fbBahn_Roll1.IsPosi_Aktiv_VonBahn:= fbGeberHandling_VonBahn_Roll1.OsAktiv;
fbBahn_Roll1.IsPosi_Fertig_VonBahn:= fbGeberHandling_VonBahn_Roll1.OsFertig
							OR	bI_AbbruchPosi_VonBahn_Roll1
								AND ( fbBahn_Roll1.SKet2 = 314
									OR	fbBahn_Roll1.SKet2 = 354
									OR	fbBahn_Roll1.SKet2 = 754
									OR	fbBahn_Roll1.SKet2 = 759 );

fbBahn_Roll1.IsLaderHatPlatteGeholt		:= strIO_GHdshk_Roll1.b_HatPlatteGeholt;
fbBahn_Roll1.IsLaderHatPlatteAbgelegt	:= strIO_GHdshk_Roll1.b_HatPlatteAbgelegt;
END_ACTION

ACTION D_Bahnjob_Riem1:
(*----------------------------------------------------------------------------------------------------------------------------------*)
(*----------------------------------------------------------------------------------------------------------------------------------*)
(*	Wenn das Bahnmodul den Job übernommen hat und der Job ausgeführt wird, muss der Job gelöscht werden					*)
(*----------------------------------------------------------------------------------------------------------------------------------*)
(*----------------------------------------------------------------------------------------------------------------------------------*)

fbBahn_Riem1.IwDoJob_AufBahn:= strIO_GHdshk_Riem1.str_DoJob_AufBahn;				(* Job Auf Bahn von der Struktur in den Baustein schreiben *)
fbBahn_Riem1.IwDoJob_VonBahn:= strIO_GHdshk_Riem1.str_DoJob_VonBahn;				(* Job Von Bahn von der Struktur in den Baustein schreiben *)
fbBahn_Riem1.IwAnzahlPlatten_BeiVonBahn := strIO_GHdshk_Riem1.i_AnzahlPlattenVonBahn;	(* Azahl der Platten in den Baustein geben *)

IF	fbBahn_Riem1.IwDoJob_AufBahn > eRolljobKeinJob							(* Wenn der Baustein den Job Auf Bahn ausführt, Job in der Struktur zurücksetzen *)
	AND	strIO_GHdshk_Riem1.str_JobAktiv_AufBahn = fbBahn_Riem1.IwDoJob_AufBahn		(* Aktiver Job in der Struktur angekommen *)
THEN
	strIO_GHdshk_Riem1.str_DoJob_AufBahn:= eRolljobKeinJob;
END_IF;

IF	fbBahn_Riem1.IwDoJob_VonBahn > eRolljobKeinJob							(* Wenn der Baustein den Job Auf Bahn ausführt, Job in der Struktur zurücksetzen *)
	AND	strIO_GHdshk_Riem1.str_JobAktiv_VonBahn = fbBahn_Riem1.IwDoJob_VonBahn		(* Aktiver Job in der Struktur angekommen *)
THEN
	strIO_GHdshk_Riem1.str_DoJob_VonBahn:= eRolljobKeinJob;
END_IF;


IF	(( fbBahn_Riem1.IsHand											(* Wenn Reset auf die Quellbahn gemacht wird, darf der Jobbaustein nicht buchen *)
		AND	fbBahn_Riem1.IsReset )
	OR	strIO_TrE.iReset <> 0 )
	AND NOT strIO_GHdshk_Riem1.b_JobVonBahnAbgebrochen
	AND 	strIO_GHdshk_Riem1.str_JobAktiv_VonBahn <> eRolljobKeinJob
	AND 	strIO_GHdshk_Riem1.str_JobAktiv_VonBahn <> eRolljobAnsBahnendeVorlauf
	AND 	strIO_GHdshk_Riem1.str_JobAktiv_VonBahn <> eRolljobAnBahnanfangRuecklauf
THEN
	strIO_GHdshk_Riem1.b_JobVonBahnAbgebrochen:= TRUE;
END_IF;
END_ACTION

ACTION D_Bahnjob_Riem2:
(*----------------------------------------------------------------------------------------------------------------------------------*)
(*----------------------------------------------------------------------------------------------------------------------------------*)
(*	Wenn das Bahnmodul den Job übernommen hat und der Job ausgeführt wird, muss der Job gelöscht werden					*)
(*----------------------------------------------------------------------------------------------------------------------------------*)
(*----------------------------------------------------------------------------------------------------------------------------------*)

fbBahn_Riem2.IwDoJob_AufBahn:= strIO_GHdshk_Riem2.str_DoJob_AufBahn;				(* Job Auf Bahn von der Struktur in den Baustein schreiben *)
fbBahn_Riem2.IwDoJob_VonBahn:= strIO_GHdshk_Riem2.str_DoJob_VonBahn;				(* Job Von Bahn von der Struktur in den Baustein schreiben *)
fbBahn_Riem2.IwAnzahlPlatten_BeiVonBahn := strIO_GHdshk_Riem2.i_AnzahlPlattenVonBahn;	(* Azahl der Platten in den Baustein geben *)

IF	fbBahn_Riem2.IwDoJob_AufBahn > eRolljobKeinJob							(* Wenn der Baustein den Job Auf Bahn ausführt, Job in der Struktur zurücksetzen *)
	AND	strIO_GHdshk_Riem2.str_JobAktiv_AufBahn = fbBahn_Riem2.IwDoJob_AufBahn		(* Aktiver Job in der Struktur angekommen *)
THEN
	strIO_GHdshk_Riem2.str_DoJob_AufBahn:= eRolljobKeinJob;
END_IF;

IF	fbBahn_Riem2.IwDoJob_VonBahn > eRolljobKeinJob							(* Wenn der Baustein den Job Auf Bahn ausführt, Job in der Struktur zurücksetzen *)
	AND	strIO_GHdshk_Riem2.str_JobAktiv_VonBahn = fbBahn_Riem2.IwDoJob_VonBahn		(* Aktiver Job in der Struktur angekommen *)
THEN
	strIO_GHdshk_Riem2.str_DoJob_VonBahn:= eRolljobKeinJob;
END_IF;


IF	(( fbBahn_Riem2.IsHand											(* Wenn Reset auf die Quellbahn gemacht wird, darf der Jobbaustein nicht buchen *)
		AND	fbBahn_Riem2.IsReset )
	OR	strIO_TrE.iReset <> 0 )
	AND NOT strIO_GHdshk_Riem2.b_JobVonBahnAbgebrochen
	AND 	strIO_GHdshk_Riem2.str_JobAktiv_VonBahn <> eRolljobKeinJob
	AND 	strIO_GHdshk_Riem2.str_JobAktiv_VonBahn <> eRolljobAnsBahnendeVorlauf
	AND 	strIO_GHdshk_Riem2.str_JobAktiv_VonBahn <> eRolljobAnBahnanfangRuecklauf
THEN
	strIO_GHdshk_Riem2.b_JobVonBahnAbgebrochen:= TRUE;
END_IF;
END_ACTION

ACTION D_Bahnjob_Roll1:
(*----------------------------------------------------------------------------------------------------------------------------------*)
(*----------------------------------------------------------------------------------------------------------------------------------*)
(*	Wenn das Bahnmodul den Job übernommen hat und der Job ausgeführt wird, muss der Job gelöscht werden					*)
(*----------------------------------------------------------------------------------------------------------------------------------*)
(*----------------------------------------------------------------------------------------------------------------------------------*)

fbBahn_Roll1.IwDoJob_AufBahn:= strIO_GHdshk_Roll1.str_DoJob_AufBahn;				(* Job Auf Bahn von der Struktur in den Baustein schreiben *)
fbBahn_Roll1.IwDoJob_VonBahn:= strIO_GHdshk_Roll1.str_DoJob_VonBahn;				(* Job Von Bahn von der Struktur in den Baustein schreiben *)
fbBahn_Roll1.IwAnzahlPlatten_BeiVonBahn:= strIO_GHdshk_Roll1.i_AnzahlPlattenVonBahn;	(* Azahl der Platten in den Baustein geben *)

IF	fbBahn_Roll1.IwDoJob_AufBahn > eRolljobKeinJob							(* Wenn der Baustein den Job Auf Bahn ausführt, Job in der Struktur zurücksetzen *)
	AND	strIO_GHdshk_Roll1.str_JobAktiv_AufBahn = fbBahn_Roll1.IwDoJob_AufBahn		(* Aktiver Job in der Struktur angekommen *)
THEN
	strIO_GHdshk_Roll1.str_DoJob_AufBahn:= eRolljobKeinJob;
END_IF;

IF	fbBahn_Roll1.IwDoJob_VonBahn > eRolljobKeinJob							(* Wenn der Baustein den Job Auf Bahn ausführt, Job in der Struktur zurücksetzen *)
	AND	strIO_GHdshk_Roll1.str_JobAktiv_VonBahn = fbBahn_Roll1.IwDoJob_VonBahn		(* Aktiver Job in der Struktur angekommen *)
THEN
	strIO_GHdshk_Roll1.str_DoJob_VonBahn:= eRolljobKeinJob;
END_IF;


IF	(( fbBahn_Roll1.IsHand											(* Wenn Reset auf die Quellbahn gemacht wird, darf der Jobbaustein nicht buchen *)
		AND	fbBahn_Roll1.IsReset )
	OR	strIO_TrE.iReset <> 0 )
	AND NOT strIO_GHdshk_Roll1.b_JobVonBahnAbgebrochen
	AND 	strIO_GHdshk_Roll1.str_JobAktiv_VonBahn <> eRolljobKeinJob
	AND 	strIO_GHdshk_Roll1.str_JobAktiv_VonBahn <> eRolljobAnsBahnendeVorlauf
	AND 	strIO_GHdshk_Roll1.str_JobAktiv_VonBahn <> eRolljobAnBahnanfangRuecklauf
THEN
	strIO_GHdshk_Roll1.b_JobVonBahnAbgebrochen:= TRUE;
END_IF;
END_ACTION

ACTION E_Ausgaenge_Hub:
(*----------------------------------------------------------------------------------------------------------------------------------*)
(*----------------------------------------------------------------------------------------------------------------------------------*)
(*                 Ausgänge Hub Winkeluebergabe															*)
(*----------------------------------------------------------------------------------------------------------------------------------*)
(*----------------------------------------------------------------------------------------------------------------------------------*)

IF	bI_Automatik
THEN
	IF	strIO_GHdshk_Riem1.b_SektionenKoppelnInY
	THEN
		bQ_Sektion1AS:= bQ_Sektion2AS;
		bQ_Sektion1GS:= bQ_Sektion2GS;

	ELSIF	fbBahn_Roll1.OwBahnStatus = iAutomatikAktivJob
	THEN
		IF	bI_HebenSenkenInvers
		THEN
			bQ_Sektion1AS:= fbBahn_Roll1.OsBahnAufFoerderhoehe;
			bQ_Sektion1GS:= NOT fbBahn_Roll1.OsBahnAufFoerderhoehe;
		ELSE
			bQ_Sektion1AS:= NOT fbBahn_Roll1.OsBahnAufFoerderhoehe;
			bQ_Sektion1GS:= fbBahn_Roll1.OsBahnAufFoerderhoehe;
		END_IF;

	ELSIF	fbBahn_Riem1.OwBahnStatus = iAutomatikAktivJob
	THEN
		IF	bI_HebenSenkenInvers
		THEN
			bQ_Sektion1AS:= NOT fbBahn_Riem1.OsBahnAufFoerderhoehe;
			bQ_Sektion1GS:= fbBahn_Riem1.OsBahnAufFoerderhoehe;
		ELSE
			bQ_Sektion1AS:= fbBahn_Riem1.OsBahnAufFoerderhoehe;
			bQ_Sektion1GS:= NOT fbBahn_Riem1.OsBahnAufFoerderhoehe;
		END_IF;
	END_IF;

	IF	strIO_GHdshk_Riem2.b_SektionenKoppelnInY
	THEN
		bQ_Sektion2AS:= bQ_Sektion1AS;
		bQ_Sektion2GS:= bQ_Sektion1GS;

	ELSIF	fbBahn_Roll1.OwBahnStatus = iAutomatikAktivJob
	THEN
		IF	bI_HebenSenkenInvers
		THEN
			bQ_Sektion2AS:= fbBahn_Roll1.OsBahnAufFoerderhoehe;
			bQ_Sektion2GS:= NOT fbBahn_Roll1.OsBahnAufFoerderhoehe;
		ELSE
			bQ_Sektion2AS:= NOT fbBahn_Roll1.OsBahnAufFoerderhoehe;
			bQ_Sektion2GS:= fbBahn_Roll1.OsBahnAufFoerderhoehe;
		END_IF;

	ELSIF	fbBahn_Riem2.OwBahnStatus = iAutomatikAktivJob
	THEN
		IF	bI_HebenSenkenInvers
		THEN
			bQ_Sektion2AS:= NOT fbBahn_Riem2.OsBahnAufFoerderhoehe;
			bQ_Sektion2GS:= fbBahn_Riem2.OsBahnAufFoerderhoehe;
		ELSE
			bQ_Sektion2AS:= fbBahn_Riem2.OsBahnAufFoerderhoehe;
			bQ_Sektion2GS:= NOT fbBahn_Riem2.OsBahnAufFoerderhoehe;
		END_IF;
	END_IF;

	IF	fbBahn_Roll1.OwBahnStatus = iAutomatikBereitJob
		AND	fbBahn_Riem1.OwBahnStatus = iAutomatikBereitJob
		AND	fbBahn_Riem2.OwBahnStatus = iAutomatikBereitJob
		AND NOT strIO_GHdshk_Roll1.b_BahnBelegt
		AND NOT strIO_GHdshk_Riem1.b_BahnBelegt
		AND NOT strIO_GHdshk_Riem2.b_BahnBelegt
		AND strIO_TrE.iAnzahlPlatten = 0
		AND strIO_TrE.asBarcode[1] = ''
	THEN
		IF	bI_HubGrundWennFrei_Sek_1
		THEN
			bQ_Sektion1AS:= FALSE;
			bQ_Sektion1GS:= TRUE;

		ELSIF bI_HubArbeitWennFrei_Sek_1
		THEN
			bQ_Sektion1AS:= TRUE;
			bQ_Sektion1GS:= FALSE;
		END_IF;

		IF	bI_HubGrundWennFrei_Sek_2
		THEN
			bQ_Sektion2AS:= FALSE;
			bQ_Sektion2GS:= TRUE;

		ELSIF bI_HubArbeitWennFrei_Sek_2
		THEN
			bQ_Sektion2AS:= TRUE;
			bQ_Sektion2GS:= FALSE;
		END_IF;

	ELSIF	fbBahn_Roll1.OwBahnStatus = iAutomatikBereitJob
		AND	fbBahn_Riem1.OwBahnStatus = iAutomatikBereitJob
		AND	fbBahn_Riem2.OwBahnStatus = iAutomatikBereitJob
		AND 	strIO_GHdshk_Roll1.b_BahnBelegt
		AND 	strIO_GHdshk_Riem1.b_BahnBelegt
		AND 	strIO_GHdshk_Riem2.b_BahnBelegt
		AND 	strIO_TrE.iAnzahlPlatten = 0
		AND 	strIO_TrE.asBarcode[1] = ''
	THEN
		IF	bI_HubGrundWennBelegt_Sek_1
		THEN
			bQ_Sektion1AS:= FALSE;
			bQ_Sektion1GS:= TRUE;

		ELSIF bI_HubArbeitWennBelegt_Sek_1
		THEN
			bQ_Sektion1AS:= TRUE;
			bQ_Sektion1GS:= FALSE;
		END_IF;

		IF	bI_HubGrundWennBelegt_Sek_2
		THEN
			bQ_Sektion2AS:= FALSE;
			bQ_Sektion2GS:= TRUE;

		ELSIF bI_HubArbeitWennBelegt_Sek_2
		THEN
			bQ_Sektion2AS:= TRUE;
			bQ_Sektion2GS:= FALSE;
		END_IF;
	END_IF;

	bHandHebenSenkenAktiv_Sek_1:= FALSE;
	bHandHebenSenkenAktiv_Sek_2:= FALSE;

ELSIF	bI_Hand
THEN
	IF	( strIO_GLmHand.bI_Heben
		OR	strIO_GLmHand.bI_Senken )
		AND	bI_FreigabeHandHebenSenkenSek1
	THEN
		bHandHebenSenkenAktiv_Sek_1:= TRUE;
	END_IF;

	IF	( strIO_GLmHand.bI_Heben
		OR	strIO_GLmHand.bI_Senken )
		AND	bI_FreigabeHandHebenSenkenSek2
	THEN
		bHandHebenSenkenAktiv_Sek_2:= TRUE;
	END_IF;

	IF	bHandHebenSenkenAktiv_Sek_1
	THEN
		bQ_Sektion1AS:= fbBahn_Roll1.OsBahnAufFoerderhoehe;
		bQ_Sektion1GS:= NOT fbBahn_Roll1.OsBahnAufFoerderhoehe;
	END_IF;

	IF	bHandHebenSenkenAktiv_Sek_2
	THEN
		bQ_Sektion2AS:= fbBahn_Roll1.OsBahnAufFoerderhoehe;
		bQ_Sektion2GS:= NOT fbBahn_Roll1.OsBahnAufFoerderhoehe;
	END_IF;

ELSE
	bHandHebenSenkenAktiv_Sek_1:= FALSE;
	bHandHebenSenkenAktiv_Sek_2:= FALSE;
END_IF;
END_ACTION

ACTION E_Ausgaenge_Riem1:
(*----------------------------------------------------------------------------------------------------------------------------------*)
(*----------------------------------------------------------------------------------------------------------------------------------*)
(*                 Ausgänge																											*)
(*----------------------------------------------------------------------------------------------------------------------------------*)
(*----------------------------------------------------------------------------------------------------------------------------------*)
fbRampe_Riem1(
	lrI_Acceleration:= strIO_GHdshk_Riem1.str_BahnRampen.lrBeschleunigung_mms2,
	lrI_Deceleration:= strIO_GHdshk_Riem1.str_BahnRampen.lrVerzoegerung_mms2,
	lrI_FastDeceleration:= strIO_GHdshk_Riem1.str_BahnRampen.lrNotverzoegerung_mms2,
	lrI_TimeBase:= lrZyklusZeit_SPS,
	lrI_MaxVelo:= strIO_GHdshk_Riem1.str_BahnSpeed.rVmaxSpeed,
	lrI_Velocity:= fbBahn_Riem1.OwBahnSpeed,
	lrI_CoupleVelocity:= fbBahn_Riem2.OwBahnSpeed,
	lrI_CoupleAcceleration:= strIO_GHdshk_Riem2.str_BahnRampen.lrBeschleunigung_mms2,
	lrI_CoupleDeceleration:= strIO_GHdshk_Riem2.str_BahnRampen.lrVerzoegerung_mms2,
	bI_Couple:= strIO_GHdshk_Riem1.b_SektionenKoppelnInY
			AND	bI_Automatik,
	bI_Enable:= bI_SicherheitOK,
	bI_ErrorQuit:= strIO_GLmHand.bI_QuittStoerung,
	lrQ_ActVelocity=> ,
	uiQ_ErrorNumber=> , 
	iQ_AnalogueValue=> ,
	bQ_TargetVelo=> , 
	bQ_Acceleration=> ,
	bQ_Deceleration=> ,
	bQ_MovePos=> , 
	bQ_MoveNeg=> , 
	bQ_MoveNot=> ,
	bQ_Error=> );

IF	fbRampe_Riem1.bQ_MovePos
THEN
	iBahnLetzteBewegung_Sek_1:= 11;

ELSIF	fbRampe_Riem1.bQ_MoveNeg
THEN
	iBahnLetzteBewegung_Sek_1:= 12;
END_IF;
END_ACTION

ACTION E_Ausgaenge_Riem2:
(*----------------------------------------------------------------------------------------------------------------------------------*)
(*----------------------------------------------------------------------------------------------------------------------------------*)
(*                 Ausgänge																											*)
(*----------------------------------------------------------------------------------------------------------------------------------*)
(*----------------------------------------------------------------------------------------------------------------------------------*)
fbRampe_Riem2(
	lrI_Acceleration:= strIO_GHdshk_Riem2.str_BahnRampen.lrBeschleunigung_mms2,
	lrI_Deceleration:= strIO_GHdshk_Riem2.str_BahnRampen.lrVerzoegerung_mms2,
	lrI_FastDeceleration:= strIO_GHdshk_Riem2.str_BahnRampen.lrNotverzoegerung_mms2,
	lrI_TimeBase:= lrZyklusZeit_SPS,
	lrI_MaxVelo:= strIO_GHdshk_Riem2.str_BahnSpeed.rVmaxSpeed,
	lrI_Velocity:= fbBahn_Riem2.OwBahnSpeed,
	lrI_CoupleVelocity:= fbBahn_Riem1.OwBahnSpeed,
	lrI_CoupleAcceleration:= strIO_GHdshk_Riem1.str_BahnRampen.lrBeschleunigung_mms2,
	lrI_CoupleDeceleration:= strIO_GHdshk_Riem1.str_BahnRampen.lrVerzoegerung_mms2,
	bI_Couple:= strIO_GHdshk_Riem2.b_SektionenKoppelnInY
			AND	bI_Automatik,
	bI_Enable:= bI_SicherheitOK,
	bI_ErrorQuit:= strIO_GLmHand.bI_QuittStoerung,
	lrQ_ActVelocity=> ,
	uiQ_ErrorNumber=> , 
	iQ_AnalogueValue=> ,
	bQ_TargetVelo=> , 
	bQ_Acceleration=> ,
	bQ_Deceleration=> ,
	bQ_MovePos=> ,
	bQ_MoveNeg=> ,
	bQ_MoveNot=> ,
	bQ_Error=> );

IF	fbRampe_Riem2.bQ_MovePos
THEN
	iBahnLetzteBewegung_Sek_2:= 11;

ELSIF	fbRampe_Riem2.bQ_MoveNeg
THEN
	iBahnLetzteBewegung_Sek_2:= 12;
END_IF;
END_ACTION

ACTION E_Ausgaenge_Roll1:
(*----------------------------------------------------------------------------------------------------------------------------------*)
(*----------------------------------------------------------------------------------------------------------------------------------*)
(*                 Ausgänge																											*)
(*----------------------------------------------------------------------------------------------------------------------------------*)
(*----------------------------------------------------------------------------------------------------------------------------------*)
fbRampe_Roll1(
	lrI_Acceleration:= strIO_GHdshk_Roll1.str_BahnRampen.lrBeschleunigung_mms2,
	lrI_Deceleration:= strIO_GHdshk_Roll1.str_BahnRampen.lrVerzoegerung_mms2,
	lrI_FastDeceleration:= strIO_GHdshk_Roll1.str_BahnRampen.lrNotverzoegerung_mms2,
	lrI_TimeBase:= lrZyklusZeit_SPS,
	lrI_MaxVelo:= strIO_GHdshk_Roll1.str_BahnSpeed.rVmaxSpeed,
	lrI_Velocity:= fbBahn_Roll1.OwBahnSpeed,
	lrI_CoupleVelocity:= 0,
	lrI_CoupleAcceleration:= 0,
	lrI_CoupleDeceleration:= 0,
	bI_Couple:= FALSE,
	bI_Enable:= bI_SicherheitOK,
	bI_ErrorQuit:= strIO_GLmHand.bI_QuittStoerung,
	lrQ_ActVelocity=> ,
	uiQ_ErrorNumber=> ,
	iQ_AnalogueValue=> ,
	bQ_TargetVelo=> , 
	bQ_Acceleration=> , 
	bQ_Deceleration=> ,
	bQ_MovePos=> ,
	bQ_MoveNeg=> , 
	bQ_MoveNot=> ,
	bQ_Error=> );

IF	fbRampe_Roll1.bQ_MovePos
THEN
	iBahnLetzteBewegung_Sek_1:= 1;
	iBahnLetzteBewegung_Sek_2:= 1;

ELSIF	fbRampe_Roll1.bQ_MoveNeg
THEN
	iBahnLetzteBewegung_Sek_1:= 2;
	iBahnLetzteBewegung_Sek_2:= 2;
END_IF;
END_ACTION

ACTION F_Positionierung_Riem1:
(*----------------------------------------------------------------------------------------------------------------------------------*)
(*----------------------------------------------------------------------------------------------------------------------------------*)
(*                 Positionierung																	*)
(*----------------------------------------------------------------------------------------------------------------------------------*)
(*----------------------------------------------------------------------------------------------------------------------------------*)


(*------ Achse Istwertsetzen  ---------------------------------*)
IF	uiI_AxId_Riem1 <> 0
THEN
	IF	fbBahn_Riem1.IwDoJob_AufBahn = eRolljobKeinJob
		AND	fbBahn_Riem1.OwJobAktiv_AufBahn = eRolljobKeinJob
		AND	fbBahn_Riem1.IwDoJob_VonBahn = eRolljobKeinJob
		AND	fbBahn_Riem1.OwJobAktiv_VonBahn = eRolljobKeinJob
		AND	fbAxIstwert_Riem1.OwOut.eAchsStatus = eStatAchse_BereitFuerJob
		AND NOT strIO_GHdshk_Riem1.b_BahnBelegt
		AND	strIO_TrE.iAnzahlPlatten = 0
		AND	strIO_TrE.asBarcode[1] = ''
		AND NOT bIstwertSetzen_Riem1
		AND ( AxFrNc_fPosIst[uiI_AxId_Riem1] > 50000
			OR	AxFrNc_fPosIst[uiI_AxId_Riem1] < -50000 )
	THEN
		bIstwertSetzen_Riem1:= TRUE;
	END_IF;

	fbAxIstwert_Riem1.AxId:= uiI_AxId_Riem1;
	fbAxIstwert_Riem1.IwResetMode:= 0;		(* Reset Modul *)

	fbAxIstwert_Riem1.IsHand:= bI_Hand;

	fbAxIstwert_Riem1.IsResetNachNotHalt:=
		AxFrNcFehler[uiI_AxId_Riem1]
		AND 	strIO_GLmHand.bI_QuittStoerung;

	fbAxIstwert_Riem1.IsAxFrNc_Auftraglaeuft:= AxFrNcAuftraglaeuft[uiI_AxId_Riem1];
	fbAxIstwert_Riem1.IsAxFrNc_Steht:= AxFrNcSteht[uiI_AxId_Riem1];
	fbAxIstwert_Riem1.IsAxFrNc_Geeicht:= AxFrNcGeeicht[uiI_AxId_Riem1];
	fbAxIstwert_Riem1.IsAxFrNc_Fehler:= AxFrNcFehler[uiI_AxId_Riem1];
	fbAxIstwert_Riem1.IwAxFrNc_nErrorCode:= AxFrNc_nErrorCode[uiI_AxId_Riem1];
	fbAxIstwert_Riem1.IsModuloAchse:= FALSE;
	
	fbAxIstwert_Riem1.IsReset:=
		( bI_FreigabeHandVorZurueck_Riem1
			OR	bI_FreigabeReset )
		AND	strIO_GLmHand.bI_Reset;
	
	IF	bIstwertSetzen_Riem1
		AND NOT fbAxIstwert_Riem1.IsIstwertSetzen
	THEN
		fbAxIstwert_Riem1.IsIstwertSetzen:= TRUE;
		fbAxIstwert_Riem1.IwWertIstwertSetzen:= 0;
	END_IF;
	
	IF	fbAxIstwert_Riem1.IsIstwertSetzen
		AND	fbAxIstwert_Riem1.OwOut.xIstwertGesetzt
	THEN
		fbAxIstwert_Riem1.IsIstwertSetzen:= FALSE;
		bIstwertSetzen_Riem1:= FALSE;
		lrIstwert_Bahn_Riem1:= 0;
	END_IF;


		fbAxIstwert_Riem1();

(*------ Simulation Istwert  ---------------------------------*)

	IF	bI_Testbetrieb
	THEN
		IF	strIO_GHdshk_Riem1.b_BahnVor
		THEN
			lrIstwert_Bahn_Riem1:=
				lrIstwert_Bahn_Riem1
				+ ABS((( strIO_GHdshk_Riem1.lr_Bahnspeed_Vorgabe * 1000) / 60 ) * lrZyklusZeit_SPS );
	
		ELSIF strIO_GHdshk_Riem1.b_BahnZurueck
		THEN
			lrIstwert_Bahn_Riem1:=
				lrIstwert_Bahn_Riem1
				- ABS((( strIO_GHdshk_Riem1.lr_Bahnspeed_Vorgabe * 1000) / 60 ) * lrZyklusZeit_SPS );
		END_IF;
	
		AxFrNc_fPosIst[uiI_AxId_Riem1]:= LREAL_TO_REAL ( lrIstwert_Bahn_Riem1 );
	END_IF;
END_IF;

IF ( bI_Testbetrieb
	OR	bI_OhneImpulsgeber_Riem1 )
	AND	uiI_AxId_Riem1 = 0
THEN
	fbVirtuellerImpulsgeber_Riem1(
		bI_Start:= strIO_GHdshk_Riem1.b_BahnVor
				OR	strIO_GHdshk_Riem1.b_BahnZurueck,
		lrI_TimeBase:= lrZyklusZeit_SPS,
		lrI_Speed:= ABS(strIO_GHdshk_Riem1.lr_Bahnspeed_Vorgabe),
		lrI_WegProImpuls:= strIO_GHdshk_Riem1.str_Bahndaten.rWegProImpuls,
		IO_Impulse:= iIncGeberZaehler_Riem1 );
END_IF;

(*------ AufBahn Positionierung Bahn  ---------------------------------*)
IF	uiI_AxId_Riem1 <> 0
THEN
	fbGeberHandling_AufBahn_Riem1.IwMode:= 1;		(* Achse auswerten *)
	fbGeberHandling_AufBahn_Riem1.IwIstwert:= AxFrNc_fPosIst[uiI_AxId_Riem1];
	fbGeberHandling_AufBahn_Riem1.IwIncGeberZaehler:= 0;
	fbGeberHandling_AufBahn_Riem1.IwWegProImpuls:= 0;
ELSE
	fbGeberHandling_AufBahn_Riem1.IwMode:= 2;		(* Zähler auswerten *)
	fbGeberHandling_AufBahn_Riem1.IwIstwert:= 0;
	fbGeberHandling_AufBahn_Riem1.IwIncGeberZaehler:= iIncGeberZaehler_Riem1;
	fbGeberHandling_AufBahn_Riem1.IwWegProImpuls:= strIO_GHdshk_Riem1.str_Bahndaten.rWegProImpuls;
END_IF;

fbGeberHandling_AufBahn_Riem1.IsAnfangBahn:= fbBahn_Riem1.IsAnfangBahn;
fbGeberHandling_AufBahn_Riem1.IsEndeBahn:= fbBahn_Riem1.IsEndeBahn;
fbGeberHandling_AufBahn_Riem1.IsStart:= fbBahn_Riem1.OsPosi_Start_AufBahn;
fbGeberHandling_AufBahn_Riem1.IsIncGeber:=  FALSE;
fbGeberHandling_AufBahn_Riem1.IsRestwertSchreiben:= TRUE;

fbGeberHandling_AufBahn_Riem1.IsIstwertGesetzt:= FALSE;
fbGeberHandling_AufBahn_Riem1.IsImRuecklauf:=
	fbBahn_Riem1.IwDoJob_AufBahn = eRolljobAufBahnPosiRuecklauf
	OR	fbBahn_Riem1.OwJobAktiv_AufBahn = eRolljobAufBahnPosiRuecklauf;

fbGeberHandling_AufBahn_Riem1.IsPosiAufBahn:=
	fbBahn_Riem1.IwDoJob_AufBahn = eRolljobAufBahnPosiVorlauf
	OR	fbBahn_Riem1.OwJobAktiv_AufBahn = eRolljobAufBahnPosiVorlauf
	OR	fbBahn_Riem1.IwDoJob_AufBahn = eRolljobAufBahnPosiRuecklauf
	OR	fbBahn_Riem1.OwJobAktiv_AufBahn = eRolljobAufBahnPosiRuecklauf;

fbGeberHandling_AufBahn_Riem1.IsPosiVonBahn:= FALSE;

fbGeberHandling_AufBahn_Riem1.IsPosi_AufDerBahn:=
	NOT fbGeberHandling_AufBahn_Riem1.IsPosiAufBahn
	AND NOT fbGeberHandling_AufBahn_Riem1.IsPosiVonBahn;

fbGeberHandling_AufBahn_Riem1.IsTestbetrieb:= bI_Testbetrieb;
fbGeberHandling_AufBahn_Riem1.IwZielPosition:= strIO_GHdshk_Riem1.r_ZielAufBahn;
fbGeberHandling_AufBahn_Riem1 ( IO_IstwertSetzen:= gxNop );


(*------ VonBahn Positionierung Bahn  ---------------------------------*)
IF	uiI_AxId_Riem1 <> 0
THEN
	fbGeberHandling_VonBahn_Riem1.IwMode:= 1;		(* Achse auswerten *)
	fbGeberHandling_VonBahn_Riem1.IwIstwert:= AxFrNc_fPosIst[uiI_AxId_Riem1];
	fbGeberHandling_VonBahn_Riem1.IwIncGeberZaehler:= 0;
	fbGeberHandling_VonBahn_Riem1.IwWegProImpuls:= 0;
ELSE
	fbGeberHandling_VonBahn_Riem1.IwMode:= 2;		(* Zähler auswerten *)
	fbGeberHandling_VonBahn_Riem1.IwIstwert:= 0;
	fbGeberHandling_VonBahn_Riem1.IwIncGeberZaehler:= iIncGeberZaehler_Riem1;
	fbGeberHandling_VonBahn_Riem1.IwWegProImpuls:= strIO_GHdshk_Riem1.str_Bahndaten.rWegProImpuls;
END_IF;

fbGeberHandling_VonBahn_Riem1.IsAnfangBahn:= fbBahn_Riem1.IsAnfangBahn;
fbGeberHandling_VonBahn_Riem1.IsEndeBahn:= fbBahn_Riem1.IsEndeBahn;
fbGeberHandling_VonBahn_Riem1.IsStart:= fbBahn_Riem1.OsPosi_Start_VonBahn;
fbGeberHandling_VonBahn_Riem1.IsIncGeber:=  FALSE;
fbGeberHandling_VonBahn_Riem1.IsRestwertSchreiben:= TRUE;

fbGeberHandling_VonBahn_Riem1.IsIstwertGesetzt:= FALSE;
fbGeberHandling_VonBahn_Riem1.IsImRuecklauf:=
	fbBahn_Riem1.IwDoJob_VonBahn = eRolljobVonBahnPosiRuecklauf
	OR	fbBahn_Riem1.OwJobAktiv_VonBahn = eRolljobVonBahnPosiRuecklauf;

fbGeberHandling_VonBahn_Riem1.IsPosiAufBahn:= FALSE;
fbGeberHandling_VonBahn_Riem1.IsPosiVonBahn:=
	fbBahn_Riem1.IwDoJob_VonBahn = eRolljobVonBahnPosiVorlauf
	OR	fbBahn_Riem1.OwJobAktiv_VonBahn = eRolljobVonBahnPosiVorlauf
	OR	fbBahn_Riem1.IwDoJob_VonBahn = eRolljobVonBahnPosiRuecklauf
	OR	fbBahn_Riem1.OwJobAktiv_VonBahn = eRolljobVonBahnPosiRuecklauf;

fbGeberHandling_VonBahn_Riem1.IsPosi_AufDerBahn:=
	NOT fbGeberHandling_VonBahn_Riem1.IsPosiVonBahn;

fbGeberHandling_VonBahn_Riem1.IsTestbetrieb:= bI_Testbetrieb;
fbGeberHandling_VonBahn_Riem1.IwZielPosition:= strIO_GHdshk_Riem1.r_ZielVonBahn;
fbGeberHandling_VonBahn_Riem1 ( IO_IstwertSetzen:= gxNop );


(*------ Position auf der Bahn  ---------------------------------*)
IF	uiI_AxId_Riem1 <> 0
THEN
	fbGeberHandling_PosPlatte_Riem1.IwMode:= 1;		(* Achse auswerten *)
	fbGeberHandling_PosPlatte_Riem1.IwIstwert:= AxFrNc_fPosIst[uiI_AxId_Riem1];
	fbGeberHandling_PosPlatte_Riem1.IwIncGeberZaehler:= 0;
	fbGeberHandling_PosPlatte_Riem1.IwWegProImpuls:= 0;
ELSE
	fbGeberHandling_PosPlatte_Riem1.IwMode:= 2;		(* Zähler auswerten *)
	fbGeberHandling_PosPlatte_Riem1.IwIstwert:= 0;
	fbGeberHandling_PosPlatte_Riem1.IwIncGeberZaehler:= iIncGeberZaehler_Riem1;
	fbGeberHandling_PosPlatte_Riem1.IwWegProImpuls:= strIO_GHdshk_Riem1.str_Bahndaten.rWegProImpuls;
END_IF;

fbGeberHandling_PosPlatte_Riem1.IsIncGeber:= FALSE;
fbGeberHandling_PosPlatte_Riem1.IsStart:= TRUE;
fbGeberHandling_PosPlatte_Riem1 ( IO_PlattenPos:= strIO_GHdshk_Riem1.str_PlattenPos );


(*------ Kontrolle des Registerimpulses  ---------------------------------*)
fbGeberKontrolle_Riem1.iI_Mode:= 2;
fbGeberKontrolle_Riem1.iI_MaxAbweichung:= strIO_GHdshk_Riem1.str_Bahndaten.iMaxAbweichungSkalierungRegisterimpuls;
fbGeberKontrolle_Riem1.iI_IncGeberZaehler:= iIncGeberZaehler_Riem1;
fbGeberKontrolle_Riem1.lrI_Geschwindigkeit:= ABS(strIO_GHdshk_Riem1.lr_Bahnspeed_Ist);
fbGeberKontrolle_Riem1.rI_WegProImpuls:= strIO_GHdshk_Riem1.str_Bahndaten.rWegProImpuls;
fbGeberKontrolle_Riem1.bI_AntriebLaeuft:= ( strIO_GHdshk_Riem1.b_BahnVor
							OR	strIO_GHdshk_Riem1.b_BahnZurueck )
							AND	ABS(strIO_GHdshk_Riem1.lr_Bahnspeed_Vorgabe) >= 5
							AND	uiI_AxId_Riem1 = 0;

fbGeberKontrolle_Riem1.bI_Testbetrieb:= bI_Testbetrieb;
fbGeberKontrolle_Riem1.bI_IfStreckenzaehler:= FALSE;
fbGeberKontrolle_Riem1.bI_QuittStoerung:=	strIO_GLmHand.bI_QuittStoerung;

fbGeberKontrolle_Riem1.tI_LaufzeitImpuls:= strIO_GHdshk_Riem1.str_BahnZeiten.tBisFehlerRegisterimpuls;
fbGeberKontrolle_Riem1.tI_LaufzeitMessung:= strIO_GHdshk_Riem1.str_BahnZeiten.tMesslaengeSkalierungRegisterimpuls;

fbGeberKontrolle_Riem1();
END_ACTION

ACTION F_Positionierung_Riem2:
(*----------------------------------------------------------------------------------------------------------------------------------*)
(*----------------------------------------------------------------------------------------------------------------------------------*)
(*                 Positionierung																	*)
(*----------------------------------------------------------------------------------------------------------------------------------*)
(*----------------------------------------------------------------------------------------------------------------------------------*)


(*------ Achse Istwertsetzen  ---------------------------------*)
IF	uiI_AxId_Riem2 <> 0
THEN
	IF	fbBahn_Riem2.IwDoJob_AufBahn = eRolljobKeinJob
		AND	fbBahn_Riem2.OwJobAktiv_AufBahn = eRolljobKeinJob
		AND	fbBahn_Riem2.IwDoJob_VonBahn = eRolljobKeinJob
		AND	fbBahn_Riem2.OwJobAktiv_VonBahn = eRolljobKeinJob
		AND	fbAxIstwert_Riem2.OwOut.eAchsStatus = eStatAchse_BereitFuerJob
		AND NOT strIO_GHdshk_Riem2.b_BahnBelegt
		AND	strIO_TrE.iAnzahlPlatten = 0
		AND	strIO_TrE.asBarcode[1] = ''
		AND NOT bIstwertSetzen_Riem2
		AND ( AxFrNc_fPosIst[uiI_AxId_Riem2] > 50000
			OR	AxFrNc_fPosIst[uiI_AxId_Riem2] < -50000 )
	THEN
		bIstwertSetzen_Riem2:= TRUE;
	END_IF;

	fbAxIstwert_Riem2.AxId:= uiI_AxId_Riem2;
	fbAxIstwert_Riem2.IwResetMode:= 0;		(* Reset Modul *)

	fbAxIstwert_Riem2.IsHand:= bI_Hand;

	fbAxIstwert_Riem2.IsResetNachNotHalt:=
		AxFrNcFehler[uiI_AxId_Riem2]
		AND 	strIO_GLmHand.bI_QuittStoerung;

	fbAxIstwert_Riem2.IsAxFrNc_Auftraglaeuft:= AxFrNcAuftraglaeuft[uiI_AxId_Riem2];
	fbAxIstwert_Riem2.IsAxFrNc_Steht:= AxFrNcSteht[uiI_AxId_Riem2];
	fbAxIstwert_Riem2.IsAxFrNc_Geeicht:= AxFrNcGeeicht[uiI_AxId_Riem2];
	fbAxIstwert_Riem2.IsAxFrNc_Fehler:= AxFrNcFehler[uiI_AxId_Riem2];
	fbAxIstwert_Riem2.IwAxFrNc_nErrorCode:= AxFrNc_nErrorCode[uiI_AxId_Riem2];
	fbAxIstwert_Riem2.IsModuloAchse:= FALSE;
	
	fbAxIstwert_Riem2.IsReset:=
		( bI_FreigabeHandVorZurueck_Riem2
			OR	bI_FreigabeReset )
		AND	strIO_GLmHand.bI_Reset;
	
	IF	bIstwertSetzen_Riem2
		AND NOT fbAxIstwert_Riem2.IsIstwertSetzen
	THEN
		fbAxIstwert_Riem2.IsIstwertSetzen:= TRUE;
		fbAxIstwert_Riem2.IwWertIstwertSetzen:= 0;
	END_IF;
	
	IF	fbAxIstwert_Riem2.IsIstwertSetzen
		AND	fbAxIstwert_Riem2.OwOut.xIstwertGesetzt
	THEN
		fbAxIstwert_Riem2.IsIstwertSetzen:= FALSE;
		bIstwertSetzen_Riem2:= FALSE;
		lrIstwert_Bahn_Riem2:= 0;
	END_IF;


		fbAxIstwert_Riem2();

(*------ Simulation Istwert  ---------------------------------*)

	IF	bI_Testbetrieb
	THEN
		IF	strIO_GHdshk_Riem2.b_BahnVor
		THEN
			lrIstwert_Bahn_Riem2:=
				lrIstwert_Bahn_Riem2
				+ ABS((( strIO_GHdshk_Riem2.lr_Bahnspeed_Vorgabe * 1000) / 60 ) * lrZyklusZeit_SPS );
	
		ELSIF strIO_GHdshk_Riem2.b_BahnZurueck
		THEN
			lrIstwert_Bahn_Riem2:=
				lrIstwert_Bahn_Riem2
				- ABS((( strIO_GHdshk_Riem2.lr_Bahnspeed_Vorgabe * 1000) / 60 ) * lrZyklusZeit_SPS );
		END_IF;
	
		AxFrNc_fPosIst[uiI_AxId_Riem2]:= LREAL_TO_REAL ( lrIstwert_Bahn_Riem2 );
	END_IF;
END_IF;

IF ( bI_Testbetrieb
	OR	bI_OhneImpulsgeber_Riem2 )
	AND	uiI_AxId_Riem2 = 0
THEN
	fbVirtuellerImpulsgeber_Riem2(
		bI_Start:= strIO_GHdshk_Riem2.b_BahnVor
				OR	strIO_GHdshk_Riem2.b_BahnZurueck,
		lrI_TimeBase:= lrZyklusZeit_SPS,
		lrI_Speed:= ABS(strIO_GHdshk_Riem2.lr_Bahnspeed_Vorgabe),
		lrI_WegProImpuls:= strIO_GHdshk_Riem2.str_Bahndaten.rWegProImpuls,
		IO_Impulse:= iIncGeberZaehler_Riem2 );
END_IF;

(*------ AufBahn Positionierung Bahn  ---------------------------------*)
IF	uiI_AxId_Riem2 <> 0
THEN
	fbGeberHandling_AufBahn_Riem2.IwMode:= 1;		(* Achse auswerten *)
	fbGeberHandling_AufBahn_Riem2.IwIstwert:= AxFrNc_fPosIst[uiI_AxId_Riem2];
	fbGeberHandling_AufBahn_Riem2.IwIncGeberZaehler:= 0;
	fbGeberHandling_AufBahn_Riem2.IwWegProImpuls:= 0;
ELSE
	fbGeberHandling_AufBahn_Riem2.IwMode:= 2;		(* Zähler auswerten *)
	fbGeberHandling_AufBahn_Riem2.IwIstwert:= 0;
	fbGeberHandling_AufBahn_Riem2.IwIncGeberZaehler:= iIncGeberZaehler_Riem2;
	fbGeberHandling_AufBahn_Riem2.IwWegProImpuls:= strIO_GHdshk_Riem2.str_Bahndaten.rWegProImpuls;
END_IF;

fbGeberHandling_AufBahn_Riem2.IsAnfangBahn:= fbBahn_Riem2.IsAnfangBahn;
fbGeberHandling_AufBahn_Riem2.IsEndeBahn:= fbBahn_Riem2.IsEndeBahn;
fbGeberHandling_AufBahn_Riem2.IsStart:= fbBahn_Riem2.OsPosi_Start_AufBahn;
fbGeberHandling_AufBahn_Riem2.IsIncGeber:=  FALSE;
fbGeberHandling_AufBahn_Riem2.IsRestwertSchreiben:= TRUE;

fbGeberHandling_AufBahn_Riem2.IsIstwertGesetzt:= FALSE;
fbGeberHandling_AufBahn_Riem2.IsImRuecklauf:=
	fbBahn_Riem2.IwDoJob_AufBahn = eRolljobAufBahnPosiRuecklauf
	OR	fbBahn_Riem2.OwJobAktiv_AufBahn = eRolljobAufBahnPosiRuecklauf;

fbGeberHandling_AufBahn_Riem2.IsPosiAufBahn:=
	fbBahn_Riem2.IwDoJob_AufBahn = eRolljobAufBahnPosiVorlauf
	OR	fbBahn_Riem2.OwJobAktiv_AufBahn = eRolljobAufBahnPosiVorlauf
	OR	fbBahn_Riem2.IwDoJob_AufBahn = eRolljobAufBahnPosiRuecklauf
	OR	fbBahn_Riem2.OwJobAktiv_AufBahn = eRolljobAufBahnPosiRuecklauf;

fbGeberHandling_AufBahn_Riem2.IsPosiVonBahn:= FALSE;

fbGeberHandling_AufBahn_Riem2.IsPosi_AufDerBahn:=
	NOT fbGeberHandling_AufBahn_Riem2.IsPosiAufBahn
	AND NOT fbGeberHandling_AufBahn_Riem2.IsPosiVonBahn;

fbGeberHandling_AufBahn_Riem2.IsTestbetrieb:= bI_Testbetrieb;
fbGeberHandling_AufBahn_Riem2.IwZielPosition:= strIO_GHdshk_Riem2.r_ZielAufBahn;
fbGeberHandling_AufBahn_Riem2 ( IO_IstwertSetzen:= gxNop );


(*------ VonBahn Positionierung Bahn  ---------------------------------*)
IF	uiI_AxId_Riem2 <> 0
THEN
	fbGeberHandling_VonBahn_Riem2.IwMode:= 1;		(* Achse auswerten *)
	fbGeberHandling_VonBahn_Riem2.IwIstwert:= AxFrNc_fPosIst[uiI_AxId_Riem2];
	fbGeberHandling_VonBahn_Riem2.IwIncGeberZaehler:= 0;
	fbGeberHandling_VonBahn_Riem2.IwWegProImpuls:= 0;
ELSE
	fbGeberHandling_VonBahn_Riem2.IwMode:= 2;		(* Zähler auswerten *)
	fbGeberHandling_VonBahn_Riem2.IwIstwert:= 0;
	fbGeberHandling_VonBahn_Riem2.IwIncGeberZaehler:= iIncGeberZaehler_Riem2;
	fbGeberHandling_VonBahn_Riem2.IwWegProImpuls:= strIO_GHdshk_Riem2.str_Bahndaten.rWegProImpuls;
END_IF;

fbGeberHandling_VonBahn_Riem2.IsAnfangBahn:= fbBahn_Riem2.IsAnfangBahn;
fbGeberHandling_VonBahn_Riem2.IsEndeBahn:= fbBahn_Riem2.IsEndeBahn;
fbGeberHandling_VonBahn_Riem2.IsStart:= fbBahn_Riem2.OsPosi_Start_VonBahn;
fbGeberHandling_VonBahn_Riem2.IsIncGeber:=  FALSE;
fbGeberHandling_VonBahn_Riem2.IsRestwertSchreiben:= TRUE;

fbGeberHandling_VonBahn_Riem2.IsIstwertGesetzt:= FALSE;
fbGeberHandling_VonBahn_Riem2.IsImRuecklauf:=
	fbBahn_Riem2.IwDoJob_VonBahn = eRolljobVonBahnPosiRuecklauf
	OR	fbBahn_Riem2.OwJobAktiv_VonBahn = eRolljobVonBahnPosiRuecklauf;

fbGeberHandling_VonBahn_Riem2.IsPosiAufBahn:= FALSE;
fbGeberHandling_VonBahn_Riem2.IsPosiVonBahn:=
	fbBahn_Riem2.IwDoJob_VonBahn = eRolljobVonBahnPosiVorlauf
	OR	fbBahn_Riem2.OwJobAktiv_VonBahn = eRolljobVonBahnPosiVorlauf
	OR	fbBahn_Riem2.IwDoJob_VonBahn = eRolljobVonBahnPosiRuecklauf
	OR	fbBahn_Riem2.OwJobAktiv_VonBahn = eRolljobVonBahnPosiRuecklauf;

fbGeberHandling_VonBahn_Riem2.IsPosi_AufDerBahn:=
	NOT fbGeberHandling_VonBahn_Riem2.IsPosiVonBahn;

fbGeberHandling_VonBahn_Riem2.IsTestbetrieb:= bI_Testbetrieb;
fbGeberHandling_VonBahn_Riem2.IwZielPosition:= strIO_GHdshk_Riem2.r_ZielVonBahn;
fbGeberHandling_VonBahn_Riem2 ( IO_IstwertSetzen:= gxNop );


(*------ Position auf der Bahn  ---------------------------------*)
IF	uiI_AxId_Riem2 <> 0
THEN
	fbGeberHandling_PosPlatte_Riem2.IwMode:= 1;		(* Achse auswerten *)
	fbGeberHandling_PosPlatte_Riem2.IwIstwert:= AxFrNc_fPosIst[uiI_AxId_Riem2];
	fbGeberHandling_PosPlatte_Riem2.IwIncGeberZaehler:= 0;
	fbGeberHandling_PosPlatte_Riem2.IwWegProImpuls:= 0;
ELSE
	fbGeberHandling_PosPlatte_Riem2.IwMode:= 2;		(* Zähler auswerten *)
	fbGeberHandling_PosPlatte_Riem2.IwIstwert:= 0;
	fbGeberHandling_PosPlatte_Riem2.IwIncGeberZaehler:= iIncGeberZaehler_Riem2;
	fbGeberHandling_PosPlatte_Riem2.IwWegProImpuls:= strIO_GHdshk_Riem2.str_Bahndaten.rWegProImpuls;
END_IF;

fbGeberHandling_PosPlatte_Riem2.IsIncGeber:= FALSE;
fbGeberHandling_PosPlatte_Riem2.IsStart:= TRUE;
fbGeberHandling_PosPlatte_Riem2 ( IO_PlattenPos:= strIO_GHdshk_Riem2.str_PlattenPos );


(*------ Kontrolle des Registerimpulses  ---------------------------------*)
fbGeberKontrolle_Riem2.iI_Mode:= 2;
fbGeberKontrolle_Riem2.iI_MaxAbweichung:= strIO_GHdshk_Riem2.str_Bahndaten.iMaxAbweichungSkalierungRegisterimpuls;
fbGeberKontrolle_Riem2.iI_IncGeberZaehler:= iIncGeberZaehler_Riem2;
fbGeberKontrolle_Riem2.lrI_Geschwindigkeit:= ABS(strIO_GHdshk_Riem2.lr_Bahnspeed_Ist);
fbGeberKontrolle_Riem2.rI_WegProImpuls:= strIO_GHdshk_Riem2.str_Bahndaten.rWegProImpuls;
fbGeberKontrolle_Riem2.bI_AntriebLaeuft:= ( strIO_GHdshk_Riem2.b_BahnVor
							OR	strIO_GHdshk_Riem2.b_BahnZurueck )
							AND	ABS(strIO_GHdshk_Riem2.lr_Bahnspeed_Vorgabe) >= 5
							AND	uiI_AxId_Riem2 = 0;

fbGeberKontrolle_Riem2.bI_Testbetrieb:= bI_Testbetrieb;
fbGeberKontrolle_Riem2.bI_IfStreckenzaehler:= FALSE;
fbGeberKontrolle_Riem2.bI_QuittStoerung:=	strIO_GLmHand.bI_QuittStoerung;

fbGeberKontrolle_Riem2.tI_LaufzeitImpuls:= strIO_GHdshk_Riem2.str_BahnZeiten.tBisFehlerRegisterimpuls;
fbGeberKontrolle_Riem2.tI_LaufzeitMessung:= strIO_GHdshk_Riem2.str_BahnZeiten.tMesslaengeSkalierungRegisterimpuls;

fbGeberKontrolle_Riem2();
END_ACTION

ACTION F_Positionierung_Roll1:
(*----------------------------------------------------------------------------------------------------------------------------------*)
(*----------------------------------------------------------------------------------------------------------------------------------*)
(*                 Positionierung																	*)
(*----------------------------------------------------------------------------------------------------------------------------------*)
(*----------------------------------------------------------------------------------------------------------------------------------*)


(*------ Achse Istwertsetzen  ---------------------------------*)
IF	uiI_AxId_Roll1 <> 0
THEN
	IF	fbBahn_Roll1.IwDoJob_AufBahn = eRolljobKeinJob
		AND	fbBahn_Roll1.OwJobAktiv_AufBahn = eRolljobKeinJob
		AND	fbBahn_Roll1.IwDoJob_VonBahn = eRolljobKeinJob
		AND	fbBahn_Roll1.OwJobAktiv_VonBahn = eRolljobKeinJob
		AND	fbAxIstwert_Roll1.OwOut.eAchsStatus = eStatAchse_BereitFuerJob
		AND NOT strIO_GHdshk_Roll1.b_BahnBelegt
		AND	strIO_TrE.iAnzahlPlatten = 0
		AND	strIO_TrE.asBarcode[1] = ''
		AND NOT bIstwertSetzen_Roll1
		AND ( AxFrNc_fPosIst[uiI_AxId_Roll1] > 50000
			OR	AxFrNc_fPosIst[uiI_AxId_Roll1] < -50000 )
	THEN
		bIstwertSetzen_Roll1:= TRUE;
	END_IF;

	fbAxIstwert_Roll1.AxId:= uiI_AxId_Roll1;
	fbAxIstwert_Roll1.IwResetMode:= 0;		(* Reset Modul *)

	fbAxIstwert_Roll1.IsHand:= bI_Hand;

	fbAxIstwert_Roll1.IsResetNachNotHalt:=
		AxFrNcFehler[uiI_AxId_Roll1]
		AND 	strIO_GLmHand.bI_QuittStoerung;

	fbAxIstwert_Roll1.IsAxFrNc_Auftraglaeuft:= AxFrNcAuftraglaeuft[uiI_AxId_Roll1];
	fbAxIstwert_Roll1.IsAxFrNc_Steht:= AxFrNcSteht[uiI_AxId_Roll1];
	fbAxIstwert_Roll1.IsAxFrNc_Geeicht:= AxFrNcGeeicht[uiI_AxId_Roll1];
	fbAxIstwert_Roll1.IsAxFrNc_Fehler:= AxFrNcFehler[uiI_AxId_Roll1];
	fbAxIstwert_Roll1.IwAxFrNc_nErrorCode:= AxFrNc_nErrorCode[uiI_AxId_Roll1];
	fbAxIstwert_Roll1.IsModuloAchse:= FALSE;
	
	fbAxIstwert_Roll1.IsReset:=
		( bI_FreigabeHandVorZurueck_Roll1
			OR	bI_FreigabeReset )
		AND	strIO_GLmHand.bI_Reset;
	
	IF	bIstwertSetzen_Roll1
		AND NOT fbAxIstwert_Roll1.IsIstwertSetzen
	THEN
		fbAxIstwert_Roll1.IsIstwertSetzen:= TRUE;
		fbAxIstwert_Roll1.IwWertIstwertSetzen:= 0;
	END_IF;
	
	IF	fbAxIstwert_Roll1.IsIstwertSetzen
		AND	fbAxIstwert_Roll1.OwOut.xIstwertGesetzt
	THEN
		fbAxIstwert_Roll1.IsIstwertSetzen:= FALSE;
		bIstwertSetzen_Roll1:= FALSE;
		lrIstwert_Bahn_Roll1:= 0;
	END_IF;


		fbAxIstwert_Roll1();

(*------ Simulation Istwert  ---------------------------------*)

	IF	bI_Testbetrieb
	THEN
		IF	strIO_GHdshk_Roll1.b_BahnVor
		THEN
			lrIstwert_Bahn_Roll1:=
				lrIstwert_Bahn_Roll1
				+ ABS((( strIO_GHdshk_Roll1.lr_Bahnspeed_Vorgabe * 1000) / 60 ) * lrZyklusZeit_SPS );
	
		ELSIF	strIO_GHdshk_Roll1.b_BahnZurueck
		THEN
			lrIstwert_Bahn_Roll1:=
				lrIstwert_Bahn_Roll1
				- ABS((( strIO_GHdshk_Roll1.lr_Bahnspeed_Vorgabe * 1000) / 60 ) * lrZyklusZeit_SPS );
		END_IF;
	
		AxFrNc_fPosIst[uiI_AxId_Roll1]:= LREAL_TO_REAL ( lrIstwert_Bahn_Roll1 );
	END_IF;
END_IF;

IF ( bI_Testbetrieb
	OR	bI_OhneImpulsgeber_Roll1 )
	AND	uiI_AxId_Roll1 = 0
THEN
	fbVirtuellerImpulsgeber_Roll1(
		bI_Start:= strIO_GHdshk_Roll1.b_BahnVor
				OR	strIO_GHdshk_Roll1.b_BahnZurueck,
		lrI_TimeBase:= lrZyklusZeit_SPS,
		lrI_Speed:= ABS(strIO_GHdshk_Roll1.lr_Bahnspeed_Vorgabe),
		lrI_WegProImpuls:= strIO_GHdshk_Roll1.str_Bahndaten.rWegProImpuls,
		IO_Impulse:= iIncGeberZaehler_Roll1 );
END_IF;

(*------ AufBahn Positionierung Bahn  ---------------------------------*)
IF	uiI_AxId_Roll1 <> 0
THEN
	fbGeberHandling_AufBahn_Roll1.IwMode:= 1;		(* Achse auswerten *)
	fbGeberHandling_AufBahn_Roll1.IwIstwert:= AxFrNc_fPosIst[uiI_AxId_Roll1];
	fbGeberHandling_AufBahn_Roll1.IwIncGeberZaehler:= 0;
	fbGeberHandling_AufBahn_Roll1.IwWegProImpuls:= 0;
ELSE
	fbGeberHandling_AufBahn_Roll1.IwMode:= 2;		(* Zähler auswerten *)
	fbGeberHandling_AufBahn_Roll1.IwIstwert:= 0;
	fbGeberHandling_AufBahn_Roll1.IwIncGeberZaehler:= iIncGeberZaehler_Roll1;
	fbGeberHandling_AufBahn_Roll1.IwWegProImpuls:= strIO_GHdshk_Roll1.str_Bahndaten.rWegProImpuls;
END_IF;

fbGeberHandling_AufBahn_Roll1.IsAnfangBahn:= fbBahn_Roll1.IsAnfangBahn;
fbGeberHandling_AufBahn_Roll1.IsEndeBahn:= fbBahn_Roll1.IsEndeBahn;
fbGeberHandling_AufBahn_Roll1.IsStart:= fbBahn_Roll1.OsPosi_Start_AufBahn;
fbGeberHandling_AufBahn_Roll1.IsIncGeber:=  FALSE;
fbGeberHandling_AufBahn_Roll1.IsRestwertSchreiben:= TRUE;

fbGeberHandling_AufBahn_Roll1.IsIstwertGesetzt:= FALSE;
fbGeberHandling_AufBahn_Roll1.IsImRuecklauf:=
	fbBahn_Roll1.IwDoJob_AufBahn = eRolljobAufBahnPosiRuecklauf
	OR	fbBahn_Roll1.OwJobAktiv_AufBahn = eRolljobAufBahnPosiRuecklauf;

fbGeberHandling_AufBahn_Roll1.IsPosiAufBahn:=
	fbBahn_Roll1.IwDoJob_AufBahn = eRolljobAufBahnPosiVorlauf
	OR	fbBahn_Roll1.OwJobAktiv_AufBahn = eRolljobAufBahnPosiVorlauf
	OR	fbBahn_Roll1.IwDoJob_AufBahn = eRolljobAufBahnPosiRuecklauf
	OR	fbBahn_Roll1.OwJobAktiv_AufBahn = eRolljobAufBahnPosiRuecklauf;

fbGeberHandling_AufBahn_Roll1.IsPosiVonBahn:= FALSE;

fbGeberHandling_AufBahn_Roll1.IsPosi_AufDerBahn:=
	NOT fbGeberHandling_AufBahn_Roll1.IsPosiAufBahn
	AND NOT fbGeberHandling_AufBahn_Roll1.IsPosiVonBahn;

fbGeberHandling_AufBahn_Roll1.IsTestbetrieb:= bI_Testbetrieb;
fbGeberHandling_AufBahn_Roll1.IwZielPosition:= strIO_GHdshk_Roll1.r_ZielAufBahn;
fbGeberHandling_AufBahn_Roll1 ( IO_IstwertSetzen:= gxNop );


(*------ VonBahn Positionierung Bahn  ---------------------------------*)
IF	uiI_AxId_Roll1 <> 0
THEN
	fbGeberHandling_VonBahn_Roll1.IwMode:= 1;		(* Achse auswerten *)
	fbGeberHandling_VonBahn_Roll1.IwIstwert:= AxFrNc_fPosIst[uiI_AxId_Roll1];
	fbGeberHandling_VonBahn_Roll1.IwIncGeberZaehler:= 0;
	fbGeberHandling_VonBahn_Roll1.IwWegProImpuls:= 0;
ELSE
	fbGeberHandling_VonBahn_Roll1.IwMode:= 2;		(* Zähler auswerten *)
	fbGeberHandling_VonBahn_Roll1.IwIstwert:= 0;
	fbGeberHandling_VonBahn_Roll1.IwIncGeberZaehler:= iIncGeberZaehler_Roll1;
	fbGeberHandling_VonBahn_Roll1.IwWegProImpuls:= strIO_GHdshk_Roll1.str_Bahndaten.rWegProImpuls;
END_IF;

fbGeberHandling_VonBahn_Roll1.IsAnfangBahn:= fbBahn_Roll1.IsAnfangBahn;
fbGeberHandling_VonBahn_Roll1.IsEndeBahn:= fbBahn_Roll1.IsEndeBahn;
fbGeberHandling_VonBahn_Roll1.IsStart:= fbBahn_Roll1.OsPosi_Start_VonBahn;
fbGeberHandling_VonBahn_Roll1.IsIncGeber:=  FALSE;
fbGeberHandling_VonBahn_Roll1.IsRestwertSchreiben:= TRUE;

fbGeberHandling_VonBahn_Roll1.IsIstwertGesetzt:= FALSE;
fbGeberHandling_VonBahn_Roll1.IsImRuecklauf:=
	fbBahn_Roll1.IwDoJob_VonBahn = eRolljobVonBahnPosiRuecklauf
	OR	fbBahn_Roll1.OwJobAktiv_VonBahn = eRolljobVonBahnPosiRuecklauf;

fbGeberHandling_VonBahn_Roll1.IsPosiAufBahn:= FALSE;
fbGeberHandling_VonBahn_Roll1.IsPosiVonBahn:=
	fbBahn_Roll1.IwDoJob_VonBahn = eRolljobVonBahnPosiVorlauf
	OR	fbBahn_Roll1.OwJobAktiv_VonBahn = eRolljobVonBahnPosiVorlauf
	OR	fbBahn_Roll1.IwDoJob_VonBahn = eRolljobVonBahnPosiRuecklauf
	OR	fbBahn_Roll1.OwJobAktiv_VonBahn = eRolljobVonBahnPosiRuecklauf;

fbGeberHandling_VonBahn_Roll1.IsPosi_AufDerBahn:=
	NOT fbGeberHandling_VonBahn_Roll1.IsPosiVonBahn;

fbGeberHandling_VonBahn_Roll1.IsTestbetrieb:= bI_Testbetrieb;
fbGeberHandling_VonBahn_Roll1.IwZielPosition:= strIO_GHdshk_Roll1.r_ZielVonBahn;
fbGeberHandling_VonBahn_Roll1 ( IO_IstwertSetzen:= gxNop );


(*------ Position auf der Bahn  ---------------------------------*)
IF	uiI_AxId_Roll1 <> 0
THEN
	fbGeberHandling_PosPlatte_Roll1.IwMode:= 1;		(* Achse auswerten *)
	fbGeberHandling_PosPlatte_Roll1.IwIstwert:= AxFrNc_fPosIst[uiI_AxId_Roll1];
	fbGeberHandling_PosPlatte_Roll1.IwIncGeberZaehler:= 0;
	fbGeberHandling_PosPlatte_Roll1.IwWegProImpuls:= 0;
ELSE
	fbGeberHandling_PosPlatte_Roll1.IwMode:= 2;		(* Zähler auswerten *)
	fbGeberHandling_PosPlatte_Roll1.IwIstwert:= 0;
	fbGeberHandling_PosPlatte_Roll1.IwIncGeberZaehler:= iIncGeberZaehler_Roll1;
	fbGeberHandling_PosPlatte_Roll1.IwWegProImpuls:= strIO_GHdshk_Roll1.str_Bahndaten.rWegProImpuls;
END_IF;

fbGeberHandling_PosPlatte_Roll1.IsIncGeber:= FALSE;
fbGeberHandling_PosPlatte_Roll1.IsStart:= TRUE;
fbGeberHandling_PosPlatte_Roll1 ( IO_PlattenPos:= strIO_GHdshk_Roll1.str_PlattenPos );


(*------ Kontrolle des Registerimpulses  ---------------------------------*)
fbGeberKontrolle_Roll1.iI_Mode:= 2;
fbGeberKontrolle_Roll1.iI_MaxAbweichung:= strIO_GHdshk_Roll1.str_Bahndaten.iMaxAbweichungSkalierungRegisterimpuls;
fbGeberKontrolle_Roll1.iI_IncGeberZaehler:= iIncGeberZaehler_Roll1;
fbGeberKontrolle_Roll1.lrI_Geschwindigkeit:= ABS(strIO_GHdshk_Roll1.lr_Bahnspeed_Ist);
fbGeberKontrolle_Roll1.rI_WegProImpuls:= strIO_GHdshk_Roll1.str_Bahndaten.rWegProImpuls;
fbGeberKontrolle_Roll1.bI_AntriebLaeuft:= ( strIO_GHdshk_Roll1.b_BahnVor
							OR	strIO_GHdshk_Roll1.b_BahnZurueck )
							AND	ABS(strIO_GHdshk_Roll1.lr_Bahnspeed_Vorgabe) >= 5
							AND	uiI_AxId_Roll1 = 0;

fbGeberKontrolle_Roll1.bI_Testbetrieb:= bI_Testbetrieb;
fbGeberKontrolle_Roll1.bI_IfStreckenzaehler:= FALSE;
fbGeberKontrolle_Roll1.bI_QuittStoerung:=	strIO_GLmHand.bI_QuittStoerung;

fbGeberKontrolle_Roll1.tI_LaufzeitImpuls:= strIO_GHdshk_Roll1.str_BahnZeiten.tBisFehlerRegisterimpuls;
fbGeberKontrolle_Roll1.tI_LaufzeitMessung:= strIO_GHdshk_Roll1.str_BahnZeiten.tMesslaengeSkalierungRegisterimpuls;

fbGeberKontrolle_Roll1();
END_ACTION

ACTION G_Protokoll_Riem1:
(*----------------------------------------------------------------------------------------------------------------------------------*)
(*----------------------------------------------------------------------------------------------------------------------------------*)
(*                Protokoll																		*)
(*----------------------------------------------------------------------------------------------------------------------------------*)
(*----------------------------------------------------------------------------------------------------------------------------------*)


(*
   Proto: Werte 'Fahrt in Grund'
*)
IF	fbBahn_Riem1.xFahrtInGrund
	AND NOT bProto_BahnInGrund_Riem1
THEN
	F_ProtoText4 ( uiI_ProId,
			CONCAT( fbBahn_Riem1.IwBahnName, ' - Fahrt in Grund' ),
			CONCAT( ' / iMode: ', F_BahnInGrund_Text( fbBahn_Riem1.IwBahnMode.iFahrtInGrund )),
			CONCAT( ' / Daten prüfen: ', BOOL_TO_STRING( fbBahn_Riem1.IwBahnMode.xDatenPruefen_NachGrund )),
			'' );

	bProto_BahnInGrund_Riem1:= TRUE;

ELSIF NOT fbBahn_Riem1.xFahrtInGrund
	AND	bProto_BahnInGrund_Riem1
THEN
	bProto_BahnInGrund_Riem1:= FALSE;
END_IF;

(*
   Protokollierung Zustände
*)

IF	iLast_Sket1_Riem1 <> fbBahn_Riem1.SKet1
	OR	iLast_Sket2_Riem1 <> fbBahn_Riem1.SKet2
	OR	bLast_Belegt_Riem1 <> fbBahn_Riem1.IsBelegtVorEndeBahn
	OR	bLast_Anfang_Riem1 <> fbBahn_Riem1.IsAnfangBahn
	OR	bLast_Ende_Riem1 <> fbBahn_Riem1.IsEndeBahn
	OR	bLast_Vorlauf_Riem1 <> fbBahn_Riem1.OsBahnVor
	OR	bLast_Zurueck_Riem1 <> fbBahn_Riem1.OsBahnZurueck
	OR	iLast_Speed_Riem1 <> fbBahn_Riem1.OwBahnSpeed
THEN
	iLast_Sket1_Riem1:= fbBahn_Riem1.SKet1;
	iLast_Sket2_Riem1:= fbBahn_Riem1.SKet2;
	bLast_Belegt_Riem1:= fbBahn_Riem1.IsBelegtVorEndeBahn;
	bLast_Anfang_Riem1:= fbBahn_Riem1.IsAnfangBahn;
	bLast_Ende_Riem1:= fbBahn_Riem1.IsEndeBahn;
	bLast_Vorlauf_Riem1:= fbBahn_Riem1.OsBahnVor;
	bLast_Zurueck_Riem1:= fbBahn_Riem1.OsBahnZurueck;
	iLast_Speed_Riem1:= fbBahn_Riem1.OwBahnSpeed;


	F_ProtoText8( uiI_ProId,
			CONCAT( fbBahn_Riem1.IwBahnName,
				  CONCAT( ' - Stat: ', INT_TO_STRING( strIO_TrE.iJobStatus ))),
			CONCAT( CONCAT( ' / Ske1: ', INT_TO_STRING( iLast_Sket1_Riem1 )),
				  CONCAT( ' / Ske2: ', INT_TO_STRING( iLast_Sket2_Riem1 ))),
			CONCAT( CONCAT( ' / Bel: ', INT_TO_STRING( strIO_TrE.iBelegtStatus )),
				  CONCAT( ' / Ist: ', INT_TO_STRING( strIO_TrE.iAnzahlPlatten ))),
			CONCAT( CONCAT( ' / Anfg: ', BOOL_TO_STRING( bLast_Anfang_Riem1 )),
				  CONCAT( ' / Ende: ', BOOL_TO_STRING( bLast_Ende_Riem1 ))),
			CONCAT( CONCAT( ' / Vor: ', BOOL_TO_STRING( bLast_Vorlauf_Riem1 )),
				  CONCAT( ' / Zur: ', BOOL_TO_STRING( bLast_Zurueck_Riem1 ))),
			CONCAT( CONCAT( ' / Speed: ', INT_TO_STRING( iLast_Speed_Riem1 )),
				  CONCAT( ' / PosPla: ', F_RealToString_2Nach( strIO_GHdshk_Riem1.str_PlattenPos.arPlattenPos[1] ))),
			CONCAT( CONCAT( ' / Auf: ', F_RealToString_2Nach( strIO_GHdshk_Riem1.r_ZielAufBahn )),
				  CONCAT( ' / Von: ', F_RealToString_2Nach( strIO_GHdshk_Riem1.r_ZielVonBahn ))),
			'' );
END_IF;
END_ACTION

ACTION G_Protokoll_Riem2:
(*----------------------------------------------------------------------------------------------------------------------------------*)
(*----------------------------------------------------------------------------------------------------------------------------------*)
(*                Protokoll																		*)
(*----------------------------------------------------------------------------------------------------------------------------------*)
(*----------------------------------------------------------------------------------------------------------------------------------*)


(*
   Proto: Werte 'Fahrt in Grund'
*)
IF	fbBahn_Riem2.xFahrtInGrund
	AND NOT bProto_BahnInGrund_Riem2
THEN
	F_ProtoText4 ( uiI_ProId,
			CONCAT( fbBahn_Riem2.IwBahnName, ' - Fahrt in Grund' ),
			CONCAT( ' / iMode: ', F_BahnInGrund_Text( fbBahn_Riem2.IwBahnMode.iFahrtInGrund )),
			CONCAT( ' / Daten prüfen: ', BOOL_TO_STRING( fbBahn_Riem2.IwBahnMode.xDatenPruefen_NachGrund )),
			'' );

	bProto_BahnInGrund_Riem2:= TRUE;

ELSIF NOT fbBahn_Riem2.xFahrtInGrund
	AND	bProto_BahnInGrund_Riem2
THEN
	bProto_BahnInGrund_Riem2:= FALSE;
END_IF;

(*
   Protokollierung Zustände
*)

IF	iLast_Sket1_Riem2 <> fbBahn_Riem2.SKet1
	OR	iLast_Sket2_Riem2 <> fbBahn_Riem2.SKet2
	OR	bLast_Belegt_Riem2 <> fbBahn_Riem2.IsBelegtVorEndeBahn
	OR	bLast_Anfang_Riem2 <> fbBahn_Riem2.IsAnfangBahn
	OR	bLast_Ende_Riem2 <> fbBahn_Riem2.IsEndeBahn
	OR	bLast_Vorlauf_Riem2 <> fbBahn_Riem2.OsBahnVor
	OR	bLast_Zurueck_Riem2 <> fbBahn_Riem2.OsBahnZurueck
	OR	iLast_Speed_Riem2 <> fbBahn_Riem2.OwBahnSpeed
THEN
	iLast_Sket1_Riem2:= fbBahn_Riem2.SKet1;
	iLast_Sket2_Riem2:= fbBahn_Riem2.SKet2;
	bLast_Belegt_Riem2:= fbBahn_Riem2.IsBelegtVorEndeBahn;
	bLast_Anfang_Riem2:= fbBahn_Riem2.IsAnfangBahn;
	bLast_Ende_Riem2:= fbBahn_Riem2.IsEndeBahn;
	bLast_Vorlauf_Riem2:= fbBahn_Riem2.OsBahnVor;
	bLast_Zurueck_Riem2:= fbBahn_Riem2.OsBahnZurueck;
	iLast_Speed_Riem2:= fbBahn_Riem2.OwBahnSpeed;


	F_ProtoText8( uiI_ProId,
			CONCAT( fbBahn_Riem2.IwBahnName,
				  CONCAT( ' - Stat: ', INT_TO_STRING( strIO_TrE.iJobStatus ))),
			CONCAT( CONCAT( ' / Ske1: ', INT_TO_STRING( iLast_Sket1_Riem2 )),
				  CONCAT( ' / Ske2: ', INT_TO_STRING( iLast_Sket2_Riem2 ))),
			CONCAT( CONCAT( ' / Bel: ', INT_TO_STRING( strIO_TrE.iBelegtStatus )),
				  CONCAT( ' / Ist: ', INT_TO_STRING( strIO_TrE.iAnzahlPlatten ))),
			CONCAT( CONCAT( ' / Anfg: ', BOOL_TO_STRING( bLast_Anfang_Riem2 )),
				  CONCAT( ' / Ende: ', BOOL_TO_STRING( bLast_Ende_Riem2 ))),
			CONCAT( CONCAT( ' / Vor: ', BOOL_TO_STRING( bLast_Vorlauf_Riem2 )),
				  CONCAT( ' / Zur: ', BOOL_TO_STRING( bLast_Zurueck_Riem2 ))),
			CONCAT( CONCAT( ' / Speed: ', INT_TO_STRING( iLast_Speed_Riem2 )),
				  CONCAT( ' / PosPla: ', F_RealToString_2Nach( strIO_GHdshk_Riem2.str_PlattenPos.arPlattenPos[1] ))),
			CONCAT( CONCAT( ' / Auf: ', F_RealToString_2Nach( strIO_GHdshk_Riem2.r_ZielAufBahn )),
				  CONCAT( ' / Von: ', F_RealToString_2Nach( strIO_GHdshk_Riem2.r_ZielVonBahn ))),
			'' );
END_IF;
END_ACTION

ACTION G_Protokoll_Roll1:
(*----------------------------------------------------------------------------------------------------------------------------------*)
(*----------------------------------------------------------------------------------------------------------------------------------*)
(*                Protokoll																		*)
(*----------------------------------------------------------------------------------------------------------------------------------*)
(*----------------------------------------------------------------------------------------------------------------------------------*)


(*
   Proto: Werte 'Fahrt in Grund'
*)
IF	fbBahn_Roll1.xFahrtInGrund
	AND NOT bProto_BahnInGrund_Roll1
THEN
	F_ProtoText4 ( uiI_ProId,
			CONCAT( fbBahn_Roll1.IwBahnName, ' - Fahrt in Grund' ),
			CONCAT( ' / iMode: ', F_BahnInGrund_Text( fbBahn_Roll1.IwBahnMode.iFahrtInGrund )),
			CONCAT( ' / Daten prüfen: ', BOOL_TO_STRING( fbBahn_Roll1.IwBahnMode.xDatenPruefen_NachGrund )),
			'' );

	bProto_BahnInGrund_Roll1:= TRUE;

ELSIF NOT fbBahn_Roll1.xFahrtInGrund
	AND	bProto_BahnInGrund_Roll1
THEN
	bProto_BahnInGrund_Roll1:= FALSE;
END_IF;

(*
   Protokollierung Zustände
*)

IF	iLast_Sket1_Roll1 <> fbBahn_Roll1.SKet1
	OR	iLast_Sket2_Roll1 <> fbBahn_Roll1.SKet2
	OR	bLast_Belegt_Roll1 <> fbBahn_Roll1.IsBelegtVorEndeBahn
	OR	bLast_Anfang_Roll1 <> fbBahn_Roll1.IsAnfangBahn
	OR	bLast_Ende_Roll1 <> fbBahn_Roll1.IsEndeBahn
	OR	bLast_Vorlauf_Roll1 <> fbBahn_Roll1.OsBahnVor
	OR	bLast_Zurueck_Roll1 <> fbBahn_Roll1.OsBahnZurueck
	OR	iLast_Speed_Roll1 <> fbBahn_Roll1.OwBahnSpeed
THEN
	iLast_Sket1_Roll1:= fbBahn_Roll1.SKet1;
	iLast_Sket2_Roll1:= fbBahn_Roll1.SKet2;
	bLast_Belegt_Roll1:= fbBahn_Roll1.IsBelegtVorEndeBahn;
	bLast_Anfang_Roll1:= fbBahn_Roll1.IsAnfangBahn;
	bLast_Ende_Roll1:= fbBahn_Roll1.IsEndeBahn;
	bLast_Vorlauf_Roll1:= fbBahn_Roll1.OsBahnVor;
	bLast_Zurueck_Roll1:= fbBahn_Roll1.OsBahnZurueck;
	iLast_Speed_Roll1:= fbBahn_Roll1.OwBahnSpeed;


	F_ProtoText8( uiI_ProId,
			CONCAT( fbBahn_Roll1.IwBahnName,
				  CONCAT( ' - Stat: ', INT_TO_STRING( strIO_TrE.iJobStatus ))),
			CONCAT( CONCAT( ' / Ske1: ', INT_TO_STRING( iLast_Sket1_Roll1 )),
				  CONCAT( ' / Ske2: ', INT_TO_STRING( iLast_Sket2_Roll1 ))),
			CONCAT( CONCAT( ' / Bel: ', INT_TO_STRING( strIO_TrE.iBelegtStatus )),
				  CONCAT( ' / Ist: ', INT_TO_STRING( strIO_TrE.iAnzahlPlatten ))),
			CONCAT( CONCAT( ' / Anfg: ', BOOL_TO_STRING( bLast_Anfang_Roll1 )),
				  CONCAT( ' / Ende: ', BOOL_TO_STRING( bLast_Ende_Roll1 ))),
			CONCAT( CONCAT( ' / Vor: ', BOOL_TO_STRING( bLast_Vorlauf_Roll1 )),
				  CONCAT( ' / Zur: ', BOOL_TO_STRING( bLast_Zurueck_Roll1 ))),
			CONCAT( CONCAT( ' / Speed: ', INT_TO_STRING( iLast_Speed_Roll1 )),
				  CONCAT( ' / PosPla: ', F_RealToString_2Nach( strIO_GHdshk_Roll1.str_PlattenPos.arPlattenPos[1] ))),
			CONCAT( CONCAT( ' / Auf: ', F_RealToString_2Nach( strIO_GHdshk_Roll1.r_ZielAufBahn )),
				  CONCAT( ' / Von: ', F_RealToString_2Nach( strIO_GHdshk_Roll1.r_ZielVonBahn ))),
			'' );
END_IF;
END_ACTION

ACTION H_Funktionsauswertung_Riem1:
(*
-------------------------------------------------------
-------------------------------------------------------

   Inhalt: 		Funtionsauswertung



   Belegtstatus:
	- iSektionFrei
	- iSektionBelegt
	- iBereitFuerLader
	- iSpurFertig
	- iGesperrt

   AufBahn Bereit für Job:
	-  0 = kein AufBahn Job darf aktiv sein
	-  1 = AufBahn Job darf aktiv sein
	-  3 = AufBahn Job 'AnsBahnende' darf aktiv sein
 	-  4 = AufBahn Job 'AnBahnanfang' darf aktiv sein
	- -1 = undefiniert

   VonBahn Bereit für Job:
	-  0 = kein VonBahn Job darf aktiv sein
	-  1 = VonBahn Job darf aktiv sein
	-  2 = Von Bahn Job + 'OsFreigabeAufBahn_BeiVonBahn' darf aktiv sein
	-  3 = Von Bahn Job 'AnsBahnende' darf aktiv sein
 	-  4 = Von Bahn Job 'AnBahnanfang' darf aktiv sein
	- -1 = undefiniert

-------------------------------------------------------
-------------------------------------------------------
*)
(*
-------------------------------------------------------
-------------------------------------------------------
	Funtionsauswertung Belegtstatus
-------------------------------------------------------
-------------------------------------------------------
*)

IF	F_GetBelegtStatus ( uiI_TrEId, iSektionFrei )
	AND NOT F_GetBelegtStatus ( uiI_TrEId, iSektionBelegt )
THEN
	strIO_GHdshk_Riem1.b_SektionFrei:= TRUE;
ELSE
	strIO_GHdshk_Riem1.b_SektionFrei:= FALSE;
END_IF;


IF	F_GetBelegtStatus ( uiI_TrEId, iSektionBelegt )
THEN
	strIO_GHdshk_Riem1.b_SektionBelegt:= TRUE;
ELSE
	strIO_GHdshk_Riem1.b_SektionBelegt:= FALSE;
END_IF;


IF	F_GetBelegtStatus ( uiI_TrEId, iBereitFuerLader )
THEN
	strIO_GHdshk_Riem1.b_BereitFuerLader:= TRUE;
ELSE
	strIO_GHdshk_Riem1.b_BereitFuerLader:= FALSE;
END_IF;


IF	F_GetBelegtStatus ( uiI_TrEId, iSektionVoll )
THEN
	strIO_GHdshk_Riem1.b_SektionVoll:= TRUE;
ELSE
	strIO_GHdshk_Riem1.b_SektionVoll:= FALSE;
END_IF;


IF	F_GetBelegtStatus ( uiI_TrEId, iSpurFertig )
THEN
	strIO_GHdshk_Riem1.b_SektionFertig:= TRUE;
ELSE
	strIO_GHdshk_Riem1.b_SektionFertig:= FALSE;
END_IF;


IF	strIO_TrE.iSperren.0
	AND	strIO_TrE.iSperren.1
THEN
	strIO_GHdshk_Riem1.b_SektionAllgemeinGesperrt:= TRUE;
ELSE
	strIO_GHdshk_Riem1.b_SektionAllgemeinGesperrt:= FALSE;
END_IF;

IF	F_GetBelegtStatus ( uiI_TrEId, iGesperrt )
	OR	strIO_TrE.iSperren.0
	OR	bIstwertSetzen_Riem1
THEN
	strIO_GHdshk_Riem1.b_SektionEinlaufGesperrt:= TRUE;
ELSE
	strIO_GHdshk_Riem1.b_SektionEinlaufGesperrt:= FALSE;
END_IF;

IF	strIO_TrE.iSperren.1
THEN
	strIO_GHdshk_Riem1.b_SektionAuslaufGesperrt:= TRUE;
ELSE
	strIO_GHdshk_Riem1.b_SektionAuslaufGesperrt:= FALSE;
END_IF;

(*
-------------------------------------------------------
-------------------------------------------------------
	Funtionsauswertung AufBahn Bereit für Job
-------------------------------------------------------
-------------------------------------------------------
*)


IF	F_BahnV2_BereitFuerJob ( 0, -1, strIO_GHdshk_Riem1  )		(* 0 = kein AufBahn Job darf aktiv sein *)
THEN
	strIO_GHdshk_Riem1.i_BahnV2_AufBahn_BereitFuerJob:= 0;

ELSIF	F_BahnV2_BereitFuerJob ( 1, -1, strIO_GHdshk_Riem1 )		(* 1 = AufBahn Job darf aktiv sein *)
THEN
	strIO_GHdshk_Riem1.i_BahnV2_AufBahn_BereitFuerJob:= 1;

ELSIF	F_BahnV2_BereitFuerJob ( 3, -1, strIO_GHdshk_Riem1 )		(* 3 = AufBahn Job 'AnsBahnende' darf aktiv sein *)
THEN
	strIO_GHdshk_Riem1.i_BahnV2_AufBahn_BereitFuerJob:= 3;

ELSIF	F_BahnV2_BereitFuerJob ( 4, -1, strIO_GHdshk_Riem1 )		(* 4 = AufBahn Job 'AnBahnanfang' darf aktiv sein *)
THEN
	strIO_GHdshk_Riem1.i_BahnV2_AufBahn_BereitFuerJob:= 4;
ELSE
	strIO_GHdshk_Riem1.i_BahnV2_AufBahn_BereitFuerJob:= 99;	(* 99 = undefiniert *)
END_IF

(*
-------------------------------------------------------
-------------------------------------------------------
Funtionsauswertung VonBahn Bereit für Job
-------------------------------------------------------
-------------------------------------------------------
*)


IF	F_BahnV2_BereitFuerJob ( -1, 0, strIO_GHdshk_Riem1 )		(* 0 = kein VonBahn Job darf aktiv sein *)
THEN
	strIO_GHdshk_Riem1.i_BahnV2_VonBahn_BereitFuerJob:= 0;

ELSIF	F_BahnV2_BereitFuerJob ( -1, 1, strIO_GHdshk_Riem1 )		(* 1 = VonBahn Job darf aktiv sein *)
THEN
	strIO_GHdshk_Riem1.i_BahnV2_VonBahn_BereitFuerJob:= 1;

ELSIF	F_BahnV2_BereitFuerJob ( -1, 2, strIO_GHdshk_Riem1 )		(* 2 = Von Bahn Job + 'OsFreigabeAufBahn_BeiVonBahn' darf aktiv sein *)
THEN
	strIO_GHdshk_Riem1.i_BahnV2_VonBahn_BereitFuerJob:= 2;

ELSIF	F_BahnV2_BereitFuerJob ( -1, 3, strIO_GHdshk_Riem1 )		(* 3 =  Von Bahn Job 'AnsBahnende' darf aktiv sein *)
THEN
	strIO_GHdshk_Riem1.i_BahnV2_VonBahn_BereitFuerJob:= 3;

ELSIF	F_BahnV2_BereitFuerJob ( -1, 4, strIO_GHdshk_Riem1 )		(* 4 =  Von Bahn Job 'AnBahnanfang' darf aktiv sein *)
THEN
	strIO_GHdshk_Riem1.i_BahnV2_VonBahn_BereitFuerJob:= 4;
ELSE
	strIO_GHdshk_Riem1.i_BahnV2_VonBahn_BereitFuerJob:= 99;	(* 99 = undefiniert *)
END_IF;
END_ACTION

ACTION H_Funktionsauswertung_Riem2:
(*
-------------------------------------------------------
-------------------------------------------------------

   Inhalt: 		Funtionsauswertung



   Belegtstatus:
	- iSektionFrei
	- iSektionBelegt
	- iBereitFuerLader
	- iSpurFertig
	- iGesperrt

   AufBahn Bereit für Job:
	-  0 = kein AufBahn Job darf aktiv sein
	-  1 = AufBahn Job darf aktiv sein
	-  3 = AufBahn Job 'AnsBahnende' darf aktiv sein
 	-  4 = AufBahn Job 'AnBahnanfang' darf aktiv sein
	- -1 = undefiniert

   VonBahn Bereit für Job:
	-  0 = kein VonBahn Job darf aktiv sein
	-  1 = VonBahn Job darf aktiv sein
	-  2 = Von Bahn Job + 'OsFreigabeAufBahn_BeiVonBahn' darf aktiv sein
	-  3 = Von Bahn Job 'AnsBahnende' darf aktiv sein
 	-  4 = Von Bahn Job 'AnBahnanfang' darf aktiv sein
	- -1 = undefiniert

-------------------------------------------------------
-------------------------------------------------------
*)
(*
-------------------------------------------------------
-------------------------------------------------------
	Funtionsauswertung Belegtstatus
-------------------------------------------------------
-------------------------------------------------------
*)

IF	F_GetBelegtStatus ( uiI_TrEId, iSektionFrei )
	AND NOT F_GetBelegtStatus ( uiI_TrEId, iSektionBelegt )
THEN
	strIO_GHdshk_Riem2.b_SektionFrei:= TRUE;
ELSE
	strIO_GHdshk_Riem2.b_SektionFrei:= FALSE;
END_IF;


IF	F_GetBelegtStatus ( uiI_TrEId, iSektionBelegt )
THEN
	strIO_GHdshk_Riem2.b_SektionBelegt:= TRUE;
ELSE
	strIO_GHdshk_Riem2.b_SektionBelegt:= FALSE;
END_IF;


IF	F_GetBelegtStatus ( uiI_TrEId, iBereitFuerLader )
THEN
	strIO_GHdshk_Riem2.b_BereitFuerLader:= TRUE;
ELSE
	strIO_GHdshk_Riem2.b_BereitFuerLader:= FALSE;
END_IF;


IF	F_GetBelegtStatus ( uiI_TrEId, iSektionVoll )
THEN
	strIO_GHdshk_Riem2.b_SektionVoll:= TRUE;
ELSE
	strIO_GHdshk_Riem2.b_SektionVoll:= FALSE;
END_IF;


IF	F_GetBelegtStatus ( uiI_TrEId, iSpurFertig )
THEN
	strIO_GHdshk_Riem2.b_SektionFertig:= TRUE;
ELSE
	strIO_GHdshk_Riem2.b_SektionFertig:= FALSE;
END_IF;


IF	strIO_TrE.iSperren.0
	AND	strIO_TrE.iSperren.1
THEN
	strIO_GHdshk_Riem2.b_SektionAllgemeinGesperrt:= TRUE;
ELSE
	strIO_GHdshk_Riem2.b_SektionAllgemeinGesperrt:= FALSE;
END_IF;

IF	F_GetBelegtStatus ( uiI_TrEId, iGesperrt )
	OR	strIO_TrE.iSperren.0
	OR	bIstwertSetzen_Riem2
THEN
	strIO_GHdshk_Riem2.b_SektionEinlaufGesperrt:= TRUE;
ELSE
	strIO_GHdshk_Riem2.b_SektionEinlaufGesperrt:= FALSE;
END_IF;

IF	strIO_TrE.iSperren.1
THEN
	strIO_GHdshk_Riem2.b_SektionAuslaufGesperrt:= TRUE;
ELSE
	strIO_GHdshk_Riem2.b_SektionAuslaufGesperrt:= FALSE;
END_IF;

(*
-------------------------------------------------------
-------------------------------------------------------
	Funtionsauswertung AufBahn Bereit für Job
-------------------------------------------------------
-------------------------------------------------------
*)


IF	F_BahnV2_BereitFuerJob ( 0, -1, strIO_GHdshk_Riem2  )		(* 0 = kein AufBahn Job darf aktiv sein *)
THEN
	strIO_GHdshk_Riem2.i_BahnV2_AufBahn_BereitFuerJob:= 0;

ELSIF	F_BahnV2_BereitFuerJob ( 1, -1, strIO_GHdshk_Riem2 )		(* 1 = AufBahn Job darf aktiv sein *)
THEN
	strIO_GHdshk_Riem2.i_BahnV2_AufBahn_BereitFuerJob:= 1;

ELSIF	F_BahnV2_BereitFuerJob ( 3, -1, strIO_GHdshk_Riem2 )		(* 3 = AufBahn Job 'AnsBahnende' darf aktiv sein *)
THEN
	strIO_GHdshk_Riem2.i_BahnV2_AufBahn_BereitFuerJob:= 3;

ELSIF	F_BahnV2_BereitFuerJob ( 4, -1, strIO_GHdshk_Riem2 )		(* 4 = AufBahn Job 'AnBahnanfang' darf aktiv sein *)
THEN
	strIO_GHdshk_Riem2.i_BahnV2_AufBahn_BereitFuerJob:= 4;
ELSE
	strIO_GHdshk_Riem2.i_BahnV2_AufBahn_BereitFuerJob:= 99;	(* 99 = undefiniert *)
END_IF

(*
-------------------------------------------------------
-------------------------------------------------------
Funtionsauswertung VonBahn Bereit für Job
-------------------------------------------------------
-------------------------------------------------------
*)


IF	F_BahnV2_BereitFuerJob ( -1, 0, strIO_GHdshk_Riem2 )		(* 0 = kein VonBahn Job darf aktiv sein *)
THEN
	strIO_GHdshk_Riem2.i_BahnV2_VonBahn_BereitFuerJob:= 0;

ELSIF	F_BahnV2_BereitFuerJob ( -1, 1, strIO_GHdshk_Riem2 )		(* 1 = VonBahn Job darf aktiv sein *)
THEN
	strIO_GHdshk_Riem2.i_BahnV2_VonBahn_BereitFuerJob:= 1;

ELSIF	F_BahnV2_BereitFuerJob ( -1, 2, strIO_GHdshk_Riem2 )		(* 2 = Von Bahn Job + 'OsFreigabeAufBahn_BeiVonBahn' darf aktiv sein *)
THEN
	strIO_GHdshk_Riem2.i_BahnV2_VonBahn_BereitFuerJob:= 2;

ELSIF	F_BahnV2_BereitFuerJob ( -1, 3, strIO_GHdshk_Riem2 )		(* 3 =  Von Bahn Job 'AnsBahnende' darf aktiv sein *)
THEN
	strIO_GHdshk_Riem2.i_BahnV2_VonBahn_BereitFuerJob:= 3;

ELSIF	F_BahnV2_BereitFuerJob ( -1, 4, strIO_GHdshk_Riem2 )		(* 4 =  Von Bahn Job 'AnBahnanfang' darf aktiv sein *)
THEN
	strIO_GHdshk_Riem2.i_BahnV2_VonBahn_BereitFuerJob:= 4;
ELSE
	strIO_GHdshk_Riem2.i_BahnV2_VonBahn_BereitFuerJob:= 99;	(* 99 = undefiniert *)
END_IF;
END_ACTION

ACTION H_Funktionsauswertung_Roll1:
(*
-------------------------------------------------------
-------------------------------------------------------

   Inhalt: 		Funtionsauswertung



   Belegtstatus:
	- iSektionFrei
	- iSektionBelegt
	- iBereitFuerLader
	- iSpurFertig
	- iGesperrt

   AufBahn Bereit für Job:
	-  0 = kein AufBahn Job darf aktiv sein
	-  1 = AufBahn Job darf aktiv sein
	-  3 = AufBahn Job 'AnsBahnende' darf aktiv sein
 	-  4 = AufBahn Job 'AnBahnanfang' darf aktiv sein
	- -1 = undefiniert

   VonBahn Bereit für Job:
	-  0 = kein VonBahn Job darf aktiv sein
	-  1 = VonBahn Job darf aktiv sein
	-  2 = Von Bahn Job + 'OsFreigabeAufBahn_BeiVonBahn' darf aktiv sein
	-  3 = Von Bahn Job 'AnsBahnende' darf aktiv sein
 	-  4 = Von Bahn Job 'AnBahnanfang' darf aktiv sein
	- -1 = undefiniert

-------------------------------------------------------
-------------------------------------------------------
*)
(*
-------------------------------------------------------
-------------------------------------------------------
	Funtionsauswertung Belegtstatus
-------------------------------------------------------
-------------------------------------------------------
*)

IF	F_GetBelegtStatus ( uiI_TrEId, iSektionFrei )
	AND NOT F_GetBelegtStatus ( uiI_TrEId, iSektionBelegt )
THEN
	strIO_GHdshk_Roll1.b_SektionFrei:= TRUE;
ELSE
	strIO_GHdshk_Roll1.b_SektionFrei:= FALSE;
END_IF;


IF	F_GetBelegtStatus ( uiI_TrEId, iSektionBelegt )
THEN
	strIO_GHdshk_Roll1.b_SektionBelegt:= TRUE;
ELSE
	strIO_GHdshk_Roll1.b_SektionBelegt:= FALSE;
END_IF;


IF	F_GetBelegtStatus ( uiI_TrEId, iBereitFuerLader )
THEN
	strIO_GHdshk_Roll1.b_BereitFuerLader:= TRUE;
ELSE
	strIO_GHdshk_Roll1.b_BereitFuerLader:= FALSE;
END_IF;


IF	F_GetBelegtStatus ( uiI_TrEId, iSektionVoll )
THEN
	strIO_GHdshk_Roll1.b_SektionVoll:= TRUE;
ELSE
	strIO_GHdshk_Roll1.b_SektionVoll:= FALSE;
END_IF;


IF	F_GetBelegtStatus ( uiI_TrEId, iSpurFertig )
THEN
	strIO_GHdshk_Roll1.b_SektionFertig:= TRUE;
ELSE
	strIO_GHdshk_Roll1.b_SektionFertig:= FALSE;
END_IF;


IF	strIO_TrE.iSperren.0
	AND	strIO_TrE.iSperren.1
THEN
	strIO_GHdshk_Roll1.b_SektionAllgemeinGesperrt:= TRUE;
ELSE
	strIO_GHdshk_Roll1.b_SektionAllgemeinGesperrt:= FALSE;
END_IF;

IF	F_GetBelegtStatus ( uiI_TrEId, iGesperrt )
	OR	strIO_TrE.iSperren.0
	OR	bIstwertSetzen_Roll1
THEN
	strIO_GHdshk_Roll1.b_SektionEinlaufGesperrt:= TRUE;
ELSE
	strIO_GHdshk_Roll1.b_SektionEinlaufGesperrt:= FALSE;
END_IF;

IF	strIO_TrE.iSperren.1
THEN
	strIO_GHdshk_Roll1.b_SektionAuslaufGesperrt:= TRUE;
ELSE
	strIO_GHdshk_Roll1.b_SektionAuslaufGesperrt:= FALSE;
END_IF;

(*
-------------------------------------------------------
-------------------------------------------------------
	Funtionsauswertung AufBahn Bereit für Job
-------------------------------------------------------
-------------------------------------------------------
*)


IF	F_BahnV2_BereitFuerJob ( 0, -1, strIO_GHdshk_Roll1  )		(* 0 = kein AufBahn Job darf aktiv sein *)
THEN
	strIO_GHdshk_Roll1.i_BahnV2_AufBahn_BereitFuerJob:= 0;

ELSIF	F_BahnV2_BereitFuerJob ( 1, -1, strIO_GHdshk_Roll1 )		(* 1 = AufBahn Job darf aktiv sein *)
THEN
	strIO_GHdshk_Roll1.i_BahnV2_AufBahn_BereitFuerJob:= 1;

ELSIF	F_BahnV2_BereitFuerJob ( 3, -1, strIO_GHdshk_Roll1 )		(* 3 = AufBahn Job 'AnsBahnende' darf aktiv sein *)
THEN
	strIO_GHdshk_Roll1.i_BahnV2_AufBahn_BereitFuerJob:= 3;

ELSIF	F_BahnV2_BereitFuerJob ( 4, -1, strIO_GHdshk_Roll1 )		(* 4 = AufBahn Job 'AnBahnanfang' darf aktiv sein *)
THEN
	strIO_GHdshk_Roll1.i_BahnV2_AufBahn_BereitFuerJob:= 4;
ELSE
	strIO_GHdshk_Roll1.i_BahnV2_AufBahn_BereitFuerJob:= 99;	(* 99 = undefiniert *)
END_IF

(*
-------------------------------------------------------
-------------------------------------------------------
Funtionsauswertung VonBahn Bereit für Job
-------------------------------------------------------
-------------------------------------------------------
*)


IF	F_BahnV2_BereitFuerJob ( -1, 0, strIO_GHdshk_Roll1 )		(* 0 = kein VonBahn Job darf aktiv sein *)
THEN
	strIO_GHdshk_Roll1.i_BahnV2_VonBahn_BereitFuerJob:= 0;

ELSIF	F_BahnV2_BereitFuerJob ( -1, 1, strIO_GHdshk_Roll1 )		(* 1 = VonBahn Job darf aktiv sein *)
THEN
	strIO_GHdshk_Roll1.i_BahnV2_VonBahn_BereitFuerJob:= 1;

ELSIF	F_BahnV2_BereitFuerJob ( -1, 2, strIO_GHdshk_Roll1 )		(* 2 = Von Bahn Job + 'OsFreigabeAufBahn_BeiVonBahn' darf aktiv sein *)
THEN
	strIO_GHdshk_Roll1.i_BahnV2_VonBahn_BereitFuerJob:= 2;

ELSIF	F_BahnV2_BereitFuerJob ( -1, 3, strIO_GHdshk_Roll1 )		(* 3 =  Von Bahn Job 'AnsBahnende' darf aktiv sein *)
THEN
	strIO_GHdshk_Roll1.i_BahnV2_VonBahn_BereitFuerJob:= 3;

ELSIF	F_BahnV2_BereitFuerJob ( -1, 4, strIO_GHdshk_Roll1 )		(* 4 =  Von Bahn Job 'AnBahnanfang' darf aktiv sein *)
THEN
	strIO_GHdshk_Roll1.i_BahnV2_VonBahn_BereitFuerJob:= 4;

ELSE
	strIO_GHdshk_Roll1.i_BahnV2_VonBahn_BereitFuerJob:= 99;	(* 99 = undefiniert *)
END_IF;
END_ACTION

ACTION H_Funktionsauswertung_Verriegelung:
(*
-------------------------------------------------------
-------------------------------------------------------

   Inhalt: 		Funtionsauswertung Verriegelung


   Sind in einer Sektion die Rollen aktiv,
   werden die Riemen auf nicht bereit gesetzt und andersherum

-------------------------------------------------------
-------------------------------------------------------
*)


IF 	strIO_GHdshk_Roll1.i_BahnV2_AufBahn_BereitFuerJob <> 0
	OR	strIO_GHdshk_Roll1.i_BahnV2_VonBahn_BereitFuerJob <> 0
THEN
	strIO_GHdshk_Riem1.i_BahnV2_AufBahn_BereitFuerJob:= 99;
	strIO_GHdshk_Riem2.i_BahnV2_AufBahn_BereitFuerJob:= 99;
	strIO_GHdshk_Riem1.i_BahnV2_VonBahn_BereitFuerJob:= 99;
	strIO_GHdshk_Riem2.i_BahnV2_VonBahn_BereitFuerJob:= 99;

ELSIF strIO_GHdshk_Riem1.i_BahnV2_AufBahn_BereitFuerJob <> 0
	OR	strIO_GHdshk_Riem2.i_BahnV2_AufBahn_BereitFuerJob <> 0
	OR	strIO_GHdshk_Riem1.i_BahnV2_VonBahn_BereitFuerJob <> 0
	OR	strIO_GHdshk_Riem2.i_BahnV2_VonBahn_BereitFuerJob <> 0
THEN
	strIO_GHdshk_Roll1.i_BahnV2_AufBahn_BereitFuerJob:= 99;
	strIO_GHdshk_Roll1.i_BahnV2_VonBahn_BereitFuerJob:= 99;
END_IF;
END_ACTION

ACTION I_TrEstati_Diagnose:
(*----------------------------------------------------------------------------------------------------------------------------------*)
(*----------------------------------------------------------------------------------------------------------------------------------*)
(*                 Belegtstatus, Aktivstatus, Diagnose Auf- und Von- Bahn										*)
(*----------------------------------------------------------------------------------------------------------------------------------*)
(*----------------------------------------------------------------------------------------------------------------------------------*)

strIO_TrE.iBelegtStatus:= F_SetClearBelegtStatus ( uiI_TrEId,	iBereitFuerLader,		( strIO_GHdshk_Roll1.b_BahnBelegt
															OR	strIO_GHdshk_Riem1.b_BahnBelegt
															OR	strIO_GHdshk_Riem2.b_BahnBelegt )
															AND	strIO_GHdshk_Roll1.b_BahnSteht
															AND	strIO_GHdshk_Roll1.i_BahnV2_AufBahn_BereitFuerJob = 0
															AND	strIO_GHdshk_Roll1.i_BahnV2_VonBahn_BereitFuerJob = 0
															AND	strIO_GHdshk_Riem1.b_BahnSteht
															AND	strIO_GHdshk_Riem1.i_BahnV2_AufBahn_BereitFuerJob = 0
															AND	strIO_GHdshk_Riem1.i_BahnV2_VonBahn_BereitFuerJob = 0
															AND	strIO_GHdshk_Riem2.b_BahnSteht
															AND	strIO_GHdshk_Riem2.i_BahnV2_AufBahn_BereitFuerJob = 0
															AND	strIO_GHdshk_Riem2.i_BahnV2_VonBahn_BereitFuerJob = 0 );
strIO_TrE.iBelegtStatus:= F_SetClearBelegtStatus ( uiI_TrEId,	iSektionBelegt,		strIO_GHdshk_Roll1.b_BahnBelegt
															OR	strIO_GHdshk_Riem1.b_BahnBelegt
															OR	strIO_GHdshk_Riem2.b_BahnBelegt );
strIO_TrE.iBelegtStatus:= F_SetClearBelegtStatus ( uiI_TrEId,	iFehlerDatenAbgleich,	fbBahn_Roll1.OsFehlerDatenAbgleich
															OR	fbBahn_Riem1.OsFehlerDatenAbgleich
															OR	fbBahn_Riem2.OsFehlerDatenAbgleich );

IF	strIO_GHdshk_Roll1.str_BahnStatus = iStoerung
	OR	strIO_GHdshk_Riem1.str_BahnStatus = iStoerung
	OR	strIO_GHdshk_Riem2.str_BahnStatus = iStoerung
THEN
	strIO_TrE.iAktivStatus:= iStoerung;

ELSIF	strIO_GHdshk_Roll1.str_BahnStatus = iFahrtGrund
	OR	strIO_GHdshk_Riem1.str_BahnStatus = iFahrtGrund
	OR	strIO_GHdshk_Riem2.str_BahnStatus = iFahrtGrund
THEN
	strIO_TrE.iAktivStatus:= iFahrtGrund;

ELSIF	strIO_GHdshk_Roll1.str_BahnStatus = iHand
	OR	strIO_GHdshk_Riem1.str_BahnStatus = iHand
	OR	strIO_GHdshk_Riem2.str_BahnStatus = iHand
THEN
	strIO_TrE.iAktivStatus:= iHand;

ELSIF	strIO_GHdshk_Roll1.str_BahnStatus = iAutomatikAktivJob
	OR	strIO_GHdshk_Riem1.str_BahnStatus = iAutomatikAktivJob
	OR	strIO_GHdshk_Riem2.str_BahnStatus = iAutomatikAktivJob
THEN
	strIO_TrE.iAktivStatus:= iAutomatikAktivJob;

ELSIF	strIO_GHdshk_Roll1.str_BahnStatus = iAutomatikBereitJob
	OR	strIO_GHdshk_Riem1.str_BahnStatus = iAutomatikBereitJob
	OR	strIO_GHdshk_Riem2.str_BahnStatus = iAutomatikBereitJob
THEN
	strIO_TrE.iAktivStatus:= iAutomatikBereitJob;

ELSE
	strIO_TrE.iAktivStatus:= iUnbekannt;
END_IF;


(*----------------------------------------------------*)
(* Bahn: Vollkennung aufheben, wenn Bahn leer		*)
(*----------------------------------------------------*)
IF	( strIO_GHdshk_Roll1.b_SektionVoll
		OR	strIO_GHdshk_Riem1.b_SektionVoll
		OR	strIO_GHdshk_Riem2.b_SektionVoll )
	AND NOT strIO_GHdshk_Roll1.b_BahnBelegt
	AND NOT fbBahn_Roll1.IsMitteBahn
	AND NOT strIO_GHdshk_Riem1.b_BahnBelegt
	AND NOT fbBahn_Riem1.IsMitteBahn
	AND NOT strIO_GHdshk_Riem2.b_BahnBelegt
	AND NOT fbBahn_Riem2.IsMitteBahn
	AND	strIO_TrE.iAnzahlPlatten = 0
	AND	strIO_GHdshk_Roll1.i_BahnV2_AufBahn_BereitFuerJob = 0
	AND	strIO_GHdshk_Roll1.i_BahnV2_VonBahn_BereitFuerJob = 0
	AND	fbBahn_Roll1.OwBahnStatus <> iStoerung
	AND	strIO_GHdshk_Riem1.i_BahnV2_AufBahn_BereitFuerJob = 0
	AND	strIO_GHdshk_Riem1.i_BahnV2_VonBahn_BereitFuerJob = 0
	AND	fbBahn_Riem1.OwBahnStatus <> iStoerung
	AND	strIO_GHdshk_Riem2.i_BahnV2_AufBahn_BereitFuerJob = 0
	AND	strIO_GHdshk_Riem2.i_BahnV2_VonBahn_BereitFuerJob = 0
	AND	fbBahn_Riem2.OwBahnStatus <> iStoerung
	AND	bI_Automatik
THEN
	strIO_TrE.iBelegtStatus:= F_SetClearBelegtStatus( uiI_TrEId, iSektionVoll, FALSE );
END_IF;

(*----------------------------------------------------*)
(* Bahn: Gesperrtkennung aufheben, wenn Bahn leer	*)
(*----------------------------------------------------*)
IF	F_GetBelegtStatus ( uiI_TrEId, iGesperrt )
	AND NOT strIO_GHdshk_Roll1.b_SektionVoll
	AND NOT strIO_GHdshk_Roll1.b_BahnBelegt
	AND NOT fbBahn_Roll1.IsMitteBahn
	AND NOT strIO_GHdshk_Riem1.b_SektionVoll
	AND NOT strIO_GHdshk_Riem1.b_BahnBelegt
	AND NOT fbBahn_Riem1.IsMitteBahn
	AND NOT strIO_GHdshk_Riem2.b_SektionVoll
	AND NOT strIO_GHdshk_Riem2.b_BahnBelegt
	AND NOT fbBahn_Riem2.IsMitteBahn
	AND	strIO_TrE.iAnzahlPlatten = 0
	AND	strIO_GHdshk_Roll1.i_BahnV2_AufBahn_BereitFuerJob = 0
	AND	strIO_GHdshk_Roll1.i_BahnV2_VonBahn_BereitFuerJob = 0
	AND	fbBahn_Roll1.OwBahnStatus <> iStoerung
	AND	strIO_GHdshk_Riem1.i_BahnV2_AufBahn_BereitFuerJob = 0
	AND	strIO_GHdshk_Riem1.i_BahnV2_VonBahn_BereitFuerJob = 0
	AND	fbBahn_Riem1.OwBahnStatus <> iStoerung
	AND	strIO_GHdshk_Riem2.i_BahnV2_AufBahn_BereitFuerJob = 0
	AND	strIO_GHdshk_Riem2.i_BahnV2_VonBahn_BereitFuerJob = 0
	AND	fbBahn_Riem2.OwBahnStatus <> iStoerung
	AND	bI_Automatik
THEN
	strIO_TrE.iBelegtStatus:= F_SetClearBelegtStatus( uiI_TrEId, iGesperrt, FALSE );
END_IF;


(* Die globale Struktur für die Leuchtmelde Handtasten beschreiben *)

IF	bI_Hand
	AND bI_FreigabeHandVorZurueck_Roll1
THEN
	IF	fbBahn_Roll1.IsBahnIstAufFoerderhoehe
		AND NOT bI_VorZurueckInversHand
		OR 	bI_BahnDarfZurueckHand_Roll1
			AND	fbBahn_Roll1.IsBahnIstAufFoerderhoehe
			AND	bI_VorZurueckInversHand
	THEN
		strIO_GLmHand.bQ_Vor:= TRUE;
	END_IF;

	IF	fbBahn_Roll1.IsBahnIstAufFoerderhoehe
		AND	bI_VorZurueckInversHand
		OR 	bI_BahnDarfZurueckHand_Roll1
			AND	fbBahn_Roll1.IsBahnIstAufFoerderhoehe
			AND NOT bI_VorZurueckInversHand
	THEN
		strIO_GLmHand.bQ_Zurueck:= TRUE;
	END_IF;
END_IF;

IF	bI_Hand
	AND bI_FreigabeHandVorZurueck_Riem1
THEN
	IF	fbBahn_Riem1.IsBahnIstAufFoerderhoehe
			AND NOT bI_VorZurueckInversHand
		OR	bI_BahnDarfZurueckHand_Riem1
			AND	fbBahn_Riem1.IsBahnIstAufFoerderhoehe
			AND	bI_VorZurueckInversHand
	THEN
		strIO_GLmHand.bQ_Vor:= TRUE;
	END_IF;

	IF	fbBahn_Riem1.IsBahnIstAufFoerderhoehe
			AND bI_VorZurueckInversHand
		OR	bI_BahnDarfZurueckHand_Riem1
			AND	fbBahn_Riem1.IsBahnIstAufFoerderhoehe
			AND NOT bI_VorZurueckInversHand
	THEN
		strIO_GLmHand.bQ_Zurueck:= TRUE;
	END_IF;
END_IF;

IF	bI_Hand
	AND bI_FreigabeHandVorZurueck_Riem2
THEN
	IF	fbBahn_Riem2.IsBahnIstAufFoerderhoehe
			AND NOT bI_VorZurueckInversHand
		OR	bI_BahnDarfZurueckHand_Riem2
			AND	fbBahn_Riem2.IsBahnIstAufFoerderhoehe
			AND	bI_VorZurueckInversHand
	THEN
		strIO_GLmHand.bQ_Vor:= TRUE;
	END_IF;

	IF	fbBahn_Riem2.IsBahnIstAufFoerderhoehe
			AND bI_VorZurueckInversHand
		OR	bI_BahnDarfZurueckHand_Riem2
			AND	fbBahn_Riem2.IsBahnIstAufFoerderhoehe
			AND NOT bI_VorZurueckInversHand
	THEN
		strIO_GLmHand.bQ_Zurueck:= TRUE;
	END_IF;
END_IF;

IF	bI_Hand
	AND ( bI_FreigabeHandHebenSenkenSek1
		OR	bI_FreigabeHandHebenSenkenSek2 )
THEN
	IF NOT fbBahn_Riem1.IsBahnIstAufFoerderhoehe
		AND	bI_FreigabeHandHebenSenkenSek1
		AND NOT bI_HebenSenkenInvers
		OR	NOT fbBahn_Riem1.IsBahnIstAufFoerderhoehe
			AND	bI_FreigabeHandHebenSenkenSek1
			AND NOT bI_HebenSenkenInvers
		OR NOT fbBahn_Roll1.IsBahnIstAufFoerderhoehe
			AND 	bI_HebenSenkenInvers
	THEN
		strIO_GLmHand.bQ_Heben:= TRUE;
	END_IF;

	IF NOT fbBahn_Roll1.IsBahnIstAufFoerderhoehe
		AND NOT bI_HebenSenkenInvers
		OR NOT fbBahn_Riem1.IsBahnIstAufFoerderhoehe
			AND	bI_FreigabeHandHebenSenkenSek1
			AND 	bI_HebenSenkenInvers
		OR NOT fbBahn_Riem2.IsBahnIstAufFoerderhoehe
			AND	bI_FreigabeHandHebenSenkenSek2
			AND 	bI_HebenSenkenInvers
	THEN
		strIO_GLmHand.bQ_Senken:= TRUE;
	END_IF;
END_IF;

IF	bI_Hand
	AND	bI_FreigabeReset
	AND ( strIO_GHdshk_Roll1.i_AblaufStatus_AufBahn <> 0
		OR	strIO_GHdshk_Roll1.i_AblaufStatus_VonBahn <> 0
		OR	strIO_GHdshk_Riem1.i_AblaufStatus_AufBahn <> 0
		OR	strIO_GHdshk_Riem1.i_AblaufStatus_VonBahn <> 0
		OR	strIO_GHdshk_Riem2.i_AblaufStatus_AufBahn <> 0
		OR	strIO_GHdshk_Riem2.i_AblaufStatus_VonBahn <> 0 )
THEN
	strIO_GLmHand.bQ_Reset:= TRUE;
END_IF;
END_ACTION

ACTION Y_Struktur_Riem1:
(*----------------------------------------------------------------------------------------------------------------------------------*)
(*----------------------------------------------------------------------------------------------------------------------------------*)
(*                Struktur																		*)
(*----------------------------------------------------------------------------------------------------------------------------------*)
(*----------------------------------------------------------------------------------------------------------------------------------*)
strIO_GHdshk_Riem1.b_ExterneBahn						:= FALSE;
strIO_GHdshk_Riem1.b_LiAnfang							:= fbEntprellenAnfang_Riem1.OsSensor;
strIO_GHdshk_Riem1.b_SwAnfang							:= bSwAnfang_Riem1;
strIO_GHdshk_Riem1.b_LiVorAnfang						:= fbEntprellenVorAnfang_Riem1.OsSensor;
strIO_GHdshk_Riem1.b_SwVorAnfang						:= bSwVorAnfang_Riem1;
strIO_GHdshk_Riem1.b_LiEnde							:= fbEntprellenEnde_Riem1.OsSensor;
strIO_GHdshk_Riem1.b_SwEnde							:= bSwEnde_Riem1;
strIO_GHdshk_Riem1.b_LiVorEnde						:= fbEntprellenVorEnde_Riem1.OsSensor;
strIO_GHdshk_Riem1.b_SwVorEnde						:= bSwVorEnde_Riem1;
strIO_GHdshk_Riem1.b_LiBelegtkontrolle					:= fbEntprellenBelegtkontrolle_Riem1.OsSensor;
strIO_GHdshk_Riem1.b_BahnIstAufFoerderhoehe				:= fbBahn_Riem1.IsBahnIstAufFoerderhoehe;
strIO_GHdshk_Riem1.b_BahnVor							:= fbRampe_Riem1.bQ_MovePos;
strIO_GHdshk_Riem1.b_BahnZurueck						:= fbRampe_Riem1.bQ_MoveNeg;
strIO_GHdshk_Riem1.b_BahnSteht						:= fbRampe_Riem1.bQ_MoveNot;
strIO_GHdshk_Riem1.b_FreimeldungAnNachSektion				:= fbBahn_Riem1.OsFreimeldungAnNachSektion
												AND ( strIO_GHdshk_Riem1_Nachf.str_JobAktiv_VonBahn = eRollJobVonBahnRuecklauf
													OR	strIO_GHdshk_Riem1_Nachf.str_JobAktiv_VonBahn = eRollJobVonBahnPosiRuecklauf
													OR	strIO_GHdshk_Riem1_Nachf.b_SektionenKoppelnInX
													OR	strIO_GHdshk_Riem1_Nachf.b_SektionenKoppelnInY
													OR	strIO_GHdshk_Riem1_Nachf.b_ExterneBahn );
strIO_GHdshk_Riem1.b_FreimeldungAnVorSektion				:= fbBahn_Riem1.OsFreimeldungAnVorSektion
												AND ( strIO_GHdshk_Riem1_Vorg.str_JobAktiv_VonBahn = eRollJobVonBahnVorlauf
													OR	strIO_GHdshk_Riem1_Vorg.str_JobAktiv_VonBahn = eRollJobVonBahnPosiVorlauf
													OR	strIO_GHdshk_Riem1_Vorg.b_SektionenKoppelnInX
													OR	strIO_GHdshk_Riem1_Vorg.b_SektionenKoppelnInY
													OR	strIO_GHdshk_Riem1_Vorg.b_ExterneBahn );
strIO_GHdshk_Riem1.b_VerstandenPlatteAbgelegt				:= fbBahn_Riem1.OsVerstandenLaderPlatteAbgelegt;
strIO_GHdshk_Riem1.b_VerstandenPlatteGeholt				:= fbBahn_Riem1.OsVerstandenLaderPlatteGeholt;
strIO_GHdshk_Riem1.i_AblaufStatus_AufBahn					:= fbBahn_Riem1.OwAblaufStatus_AufBahn;
strIO_GHdshk_Riem1.i_AblaufStatus_VonBahn					:= fbBahn_Riem1.OwAblaufStatus_VonBahn;
strIO_GHdshk_Riem1.str_BahnStatus						:= fbBahn_Riem1.OwBahnStatus;
strIO_GHdshk_Riem1.str_JobAktiv_AufBahn					:= fbBahn_Riem1.OwJobAktiv_AufBahn;
strIO_GHdshk_Riem1.str_JobAktiv_VonBahn					:= fbBahn_Riem1.OwJobAktiv_VonBahn;
strIO_GHdshk_Riem1.b_MBahnBelegt_KeineDaten				:= fbBahn_Riem1.OsMBahnBelegt_KeineDaten;
strIO_GHdshk_Riem1.b_MBahnFrei_Daten					:= fbBahn_Riem1.OsMBahnFrei_Daten;
strIO_GHdshk_Riem1.b_MBahnNichtAufFoerderhoehe				:= fbBahn_Riem1.OsMBahnNichtAufFoerderhoehe;
strIO_GHdshk_Riem1.b_MMaxLaufzeit_AufBahn					:= fbBahn_Riem1.OsMMaxLaufzeit_AufBahn;
strIO_GHdshk_Riem1.b_MMaxLaufzeit_VonBahn					:= fbBahn_Riem1.OsMMaxLaufzeit_VonBahn;
strIO_GHdshk_Riem1.b_MStoerungAntrieb					:= fbBahn_Riem1.OsMStoerungAntrieb;
strIO_GHdshk_Riem1.b_MKeineFreigabe_FahrtInGrund			:= fbBahn_Riem1.OsMKeineFreigabe_FahrtInGrund;
strIO_GHdshk_Riem1.b_MFehlerRegisterimpuls				:= fbGeberKontrolle_Riem1.bQ_FehlerGeber;
strIO_GHdshk_Riem1.b_MFehlerSkalierung					:= fbGeberKontrolle_Riem1.bQ_FehlerSkalierung;

strIO_GHdshk_Riem1.b_GeberHandling_AufBahn_Aktiv			:= fbGeberHandling_AufBahn_Riem1.OsAktiv;
strIO_GHdshk_Riem1.b_GeberHandling_AufBahn_Fertig			:= fbGeberHandling_AufBahn_Riem1.OsFertig;
strIO_GHdshk_Riem1.r_PosiRestwert_AufBahn					:= fbGeberHandling_AufBahn_Riem1.OwPosiRestWert;

strIO_GHdshk_Riem1.b_GeberHandling_VonBahn_Aktiv			:= fbGeberHandling_VonBahn_Riem1.OsAktiv;
strIO_GHdshk_Riem1.b_GeberHandling_VonBahn_Fertig			:= fbGeberHandling_VonBahn_Riem1.OsFertig;
strIO_GHdshk_Riem1.r_PosiRestwert_VonBahn					:= fbGeberHandling_VonBahn_Riem1.OwPosiRestWert;

IF	fbRampe_Riem1.bI_Couple
THEN
	strIO_GHdshk_Riem1.lr_Bahnspeed_Soll				:= fbRampe_Riem1.lrI_CoupleVelocity;
ELSE
	strIO_GHdshk_Riem1.lr_Bahnspeed_Soll				:= fbRampe_Riem1.lrI_Velocity;
END_IF;

strIO_GHdshk_Riem1.lr_Bahnspeed_Vorgabe					:= fbRampe_Riem1.lrQ_ActVelocity;

IF	( strIO_GHdshk_Riem1.b_LiAnfang
	AND	strIO_GHdshk_Riem1.str_JobAktiv_AufBahn <> eRolljobAufBahnVorlauf
	AND	strIO_GHdshk_Riem1.str_JobAktiv_AufBahn <> eRolljobAufBahnPosiVorlauf
	AND	strIO_GHdshk_Riem1.b_BahnVor
	OR	strIO_GHdshk_Riem1.b_LiEnde
		AND	strIO_GHdshk_Riem1.str_JobAktiv_AufBahn <> eRolljobAufBahnRuecklauf
		AND	strIO_GHdshk_Riem1.str_JobAktiv_AufBahn <> eRolljobAufBahnPosiRuecklauf
		AND	strIO_GHdshk_Riem1.b_BahnZurueck )
	AND NOT strIO_GHdshk_Riem1.b_MTeilNichtFreigegeben
	AND NOT strIO_GLmHand.bI_QuittStoerung
	AND	bI_Automatik
	AND	bI_MitUeberwachungTeilNichtFreigegeben
THEN
	strIO_GHdshk_Riem1.b_MTeilNichtFreigegeben:= TRUE;

ELSIF	strIO_GLmHand.bI_QuittStoerung
THEN
	strIO_GHdshk_Riem1.b_MTeilNichtFreigegeben:= FALSE;
END_IF;

IF NOT strIO_GHdshk_Riem2.b_SektionenKoppelnInX				(* wenn Riem2 einfördert + andere Bahn nur 1 Sektion + Riem1 nix tut, dann die Freigaben von Riem2 in Riem1 nehmen *)
	AND NOT strIO_GHdshk_Riem2.b_SektionenKoppelnInY
	AND (( strIO_GHdshk_Riem2.str_JobAktiv_AufBahn = eRolljobAufBahnPosiVorlauf
		OR	strIO_GHdshk_Riem2.str_JobAktiv_AufBahn = eRolljobAufBahnVorlauf )
		AND	bI_VorgRiemHatNurEineSpur
		OR ( strIO_GHdshk_Riem2.str_JobAktiv_AufBahn = eRolljobAufBahnPosiRuecklauf
			OR	strIO_GHdshk_Riem2.str_JobAktiv_AufBahn = eRolljobAufBahnRuecklauf )
			AND	bI_NachfRiemHatNurEineSpur )
	AND	strIO_GHdshk_Riem1.i_BahnV2_AufBahn_BereitFuerJob = 0
	AND	strIO_GHdshk_Riem1.i_BahnV2_VonBahn_BereitFuerJob = 0
	AND	bI_Automatik
THEN
	strIO_GHdshk_Riem1.b_FreimeldungAnNachSektion			:= fbBahn_Riem2.OsFreimeldungAnNachSektion
												AND ( strIO_GHdshk_Riem1_Nachf.str_JobAktiv_VonBahn = eRollJobVonBahnRuecklauf
													OR	strIO_GHdshk_Riem1_Nachf.str_JobAktiv_VonBahn = eRollJobVonBahnPosiRuecklauf
													OR	strIO_GHdshk_Riem1_Nachf.b_SektionenKoppelnInX
													OR	strIO_GHdshk_Riem1_Nachf.b_SektionenKoppelnInY
													OR	strIO_GHdshk_Riem1_Nachf.b_ExterneBahn
													OR	bI_NachfRiemHatNurEineSpur );
	strIO_GHdshk_Riem1.b_FreimeldungAnVorSektion			:= fbBahn_Riem2.OsFreimeldungAnVorSektion
												AND ( strIO_GHdshk_Riem1_Vorg.str_JobAktiv_VonBahn = eRollJobVonBahnVorlauf
													OR	strIO_GHdshk_Riem1_Vorg.str_JobAktiv_VonBahn = eRollJobVonBahnPosiVorlauf
													OR	strIO_GHdshk_Riem1_Vorg.b_SektionenKoppelnInX
													OR	strIO_GHdshk_Riem1_Vorg.b_SektionenKoppelnInY
													OR	strIO_GHdshk_Riem1_Vorg.b_ExterneBahn
													OR	bI_VorgRiemHatNurEineSpur );

	IF	fbRampe_Riem2.bI_Couple
	THEN
		strIO_GHdshk_Riem1.lr_Bahnspeed_Soll			:= fbRampe_Riem2.lrI_CoupleVelocity;
	ELSE
		strIO_GHdshk_Riem1.lr_Bahnspeed_Soll			:= fbRampe_Riem2.lrI_Velocity;
	END_IF;

	strIO_GHdshk_Riem1.lr_Bahnspeed_Vorgabe				:= fbRampe_Riem2.lrQ_ActVelocity;
ELSE
	strIO_GHdshk_Riem1.b_FreimeldungAnNachSektion			:= fbBahn_Riem1.OsFreimeldungAnNachSektion
												AND ( strIO_GHdshk_Riem1_Nachf.str_JobAktiv_VonBahn = eRollJobVonBahnRuecklauf
													OR	strIO_GHdshk_Riem1_Nachf.str_JobAktiv_VonBahn = eRollJobVonBahnPosiRuecklauf
													OR	strIO_GHdshk_Riem1_Nachf.b_SektionenKoppelnInX
													OR	strIO_GHdshk_Riem1_Nachf.b_SektionenKoppelnInY
													OR	strIO_GHdshk_Riem1_Nachf.b_ExterneBahn );
	strIO_GHdshk_Riem1.b_FreimeldungAnVorSektion			:= fbBahn_Riem1.OsFreimeldungAnVorSektion
												AND ( strIO_GHdshk_Riem1_Vorg.str_JobAktiv_VonBahn = eRollJobVonBahnVorlauf
													OR	strIO_GHdshk_Riem1_Vorg.str_JobAktiv_VonBahn = eRollJobVonBahnPosiVorlauf
													OR	strIO_GHdshk_Riem1_Vorg.b_SektionenKoppelnInX
													OR	strIO_GHdshk_Riem1_Vorg.b_SektionenKoppelnInY
													OR	strIO_GHdshk_Riem1_Vorg.b_ExterneBahn );

	IF	fbRampe_Riem1.bI_Couple
	THEN
		strIO_GHdshk_Riem1.lr_Bahnspeed_Soll			:= fbRampe_Riem1.lrI_CoupleVelocity;
	ELSE
		strIO_GHdshk_Riem1.lr_Bahnspeed_Soll			:= fbRampe_Riem1.lrI_Velocity;
	END_IF;

	strIO_GHdshk_Riem1.lr_Bahnspeed_Vorgabe				:= fbRampe_Riem1.lrQ_ActVelocity;
END_IF;
END_ACTION

ACTION Y_Struktur_Riem2:
(*----------------------------------------------------------------------------------------------------------------------------------*)
(*----------------------------------------------------------------------------------------------------------------------------------*)
(*                Struktur																		*)
(*----------------------------------------------------------------------------------------------------------------------------------*)
(*----------------------------------------------------------------------------------------------------------------------------------*)
strIO_GHdshk_Riem2.b_ExterneBahn						:= FALSE;
strIO_GHdshk_Riem2.b_LiAnfang							:= fbEntprellenAnfang_Riem2.OsSensor;
strIO_GHdshk_Riem2.b_SwAnfang							:= bSwAnfang_Riem2;
strIO_GHdshk_Riem2.b_LiVorAnfang						:= fbEntprellenVorAnfang_Riem2.OsSensor;
strIO_GHdshk_Riem2.b_SwVorAnfang						:= bSwVorAnfang_Riem2;
strIO_GHdshk_Riem2.b_LiEnde							:= fbEntprellenEnde_Riem2.OsSensor;
strIO_GHdshk_Riem2.b_SwEnde							:= bSwEnde_Riem2;
strIO_GHdshk_Riem2.b_LiVorEnde						:= fbEntprellenVorEnde_Riem2.OsSensor;
strIO_GHdshk_Riem2.b_SwVorEnde						:= bSwVorEnde_Riem2;
strIO_GHdshk_Riem2.b_LiBelegtkontrolle					:= fbEntprellenBelegtkontrolle_Riem2.OsSensor;
strIO_GHdshk_Riem2.b_BahnIstAufFoerderhoehe				:= fbBahn_Riem2.IsBahnIstAufFoerderhoehe;
strIO_GHdshk_Riem2.b_BahnVor							:= fbRampe_Riem2.bQ_MovePos;
strIO_GHdshk_Riem2.b_BahnZurueck						:= fbRampe_Riem2.bQ_MoveNeg;
strIO_GHdshk_Riem2.b_BahnSteht						:= fbRampe_Riem2.bQ_MoveNot;
strIO_GHdshk_Riem2.b_FreimeldungAnNachSektion				:= fbBahn_Riem2.OsFreimeldungAnNachSektion
												AND ( strIO_GHdshk_Riem2_Nachf.str_JobAktiv_VonBahn = eRollJobVonBahnRuecklauf
													OR	strIO_GHdshk_Riem2_Nachf.str_JobAktiv_VonBahn = eRollJobVonBahnPosiRuecklauf
													OR	strIO_GHdshk_Riem2_Nachf.b_SektionenKoppelnInX
													OR	strIO_GHdshk_Riem2_Nachf.b_SektionenKoppelnInY
													OR	strIO_GHdshk_Riem2_Nachf.b_ExterneBahn
													OR	bI_NachfRiemHatNurEineSpur );
strIO_GHdshk_Riem2.b_FreimeldungAnVorSektion				:= fbBahn_Riem2.OsFreimeldungAnVorSektion
												AND ( strIO_GHdshk_Riem2_Vorg.str_JobAktiv_VonBahn = eRollJobVonBahnVorlauf
													OR	strIO_GHdshk_Riem2_Vorg.str_JobAktiv_VonBahn = eRollJobVonBahnPosiVorlauf
													OR	strIO_GHdshk_Riem2_Vorg.b_SektionenKoppelnInX
													OR	strIO_GHdshk_Riem2_Vorg.b_SektionenKoppelnInY
													OR	strIO_GHdshk_Riem2_Vorg.b_ExterneBahn
													OR	bI_VorgRiemHatNurEineSpur );
strIO_GHdshk_Riem2.b_VerstandenPlatteAbgelegt				:= fbBahn_Riem2.OsVerstandenLaderPlatteAbgelegt;
strIO_GHdshk_Riem2.b_VerstandenPlatteGeholt				:= fbBahn_Riem2.OsVerstandenLaderPlatteGeholt;
strIO_GHdshk_Riem2.i_AblaufStatus_AufBahn					:= fbBahn_Riem2.OwAblaufStatus_AufBahn;
strIO_GHdshk_Riem2.i_AblaufStatus_VonBahn					:= fbBahn_Riem2.OwAblaufStatus_VonBahn;
strIO_GHdshk_Riem2.str_BahnStatus						:= fbBahn_Riem2.OwBahnStatus;
strIO_GHdshk_Riem2.str_JobAktiv_AufBahn					:= fbBahn_Riem2.OwJobAktiv_AufBahn;
strIO_GHdshk_Riem2.str_JobAktiv_VonBahn					:= fbBahn_Riem2.OwJobAktiv_VonBahn;
strIO_GHdshk_Riem2.b_MBahnBelegt_KeineDaten				:= fbBahn_Riem2.OsMBahnBelegt_KeineDaten;
strIO_GHdshk_Riem2.b_MBahnFrei_Daten					:= fbBahn_Riem2.OsMBahnFrei_Daten;
strIO_GHdshk_Riem2.b_MBahnNichtAufFoerderhoehe				:= fbBahn_Riem2.OsMBahnNichtAufFoerderhoehe;
strIO_GHdshk_Riem2.b_MMaxLaufzeit_AufBahn					:= fbBahn_Riem2.OsMMaxLaufzeit_AufBahn;
strIO_GHdshk_Riem2.b_MMaxLaufzeit_VonBahn					:= fbBahn_Riem2.OsMMaxLaufzeit_VonBahn;
strIO_GHdshk_Riem2.b_MStoerungAntrieb					:= fbBahn_Riem2.OsMStoerungAntrieb;
strIO_GHdshk_Riem2.b_MKeineFreigabe_FahrtInGrund			:= fbBahn_Riem2.OsMKeineFreigabe_FahrtInGrund;
strIO_GHdshk_Riem2.b_MFehlerRegisterimpuls				:= fbGeberKontrolle_Riem2.bQ_FehlerGeber;
strIO_GHdshk_Riem2.b_MFehlerSkalierung					:= fbGeberKontrolle_Riem2.bQ_FehlerSkalierung;

strIO_GHdshk_Riem2.b_GeberHandling_AufBahn_Aktiv			:= fbGeberHandling_AufBahn_Riem2.OsAktiv;
strIO_GHdshk_Riem2.b_GeberHandling_AufBahn_Fertig			:= fbGeberHandling_AufBahn_Riem2.OsFertig;
strIO_GHdshk_Riem2.r_PosiRestwert_AufBahn					:= fbGeberHandling_AufBahn_Riem2.OwPosiRestWert;

strIO_GHdshk_Riem2.b_GeberHandling_VonBahn_Aktiv			:= fbGeberHandling_VonBahn_Riem2.OsAktiv;
strIO_GHdshk_Riem2.b_GeberHandling_VonBahn_Fertig			:= fbGeberHandling_VonBahn_Riem2.OsFertig;
strIO_GHdshk_Riem2.r_PosiRestwert_VonBahn					:= fbGeberHandling_VonBahn_Riem2.OwPosiRestWert;

IF	fbRampe_Riem2.bI_Couple
THEN
	strIO_GHdshk_Riem2.lr_Bahnspeed_Soll				:= fbRampe_Riem2.lrI_CoupleVelocity;
ELSE
	strIO_GHdshk_Riem2.lr_Bahnspeed_Soll				:= fbRampe_Riem2.lrI_Velocity;
END_IF;

strIO_GHdshk_Riem2.lr_Bahnspeed_Vorgabe					:= fbRampe_Riem2.lrQ_ActVelocity;

IF	( strIO_GHdshk_Riem2.b_LiAnfang
	AND	strIO_GHdshk_Riem2.str_JobAktiv_AufBahn <> eRolljobAufBahnVorlauf
	AND	strIO_GHdshk_Riem2.str_JobAktiv_AufBahn <> eRolljobAufBahnPosiVorlauf
	AND	strIO_GHdshk_Riem2.b_BahnVor
	OR	strIO_GHdshk_Riem2.b_LiEnde
		AND	strIO_GHdshk_Riem2.str_JobAktiv_AufBahn <> eRolljobAufBahnRuecklauf
		AND	strIO_GHdshk_Riem2.str_JobAktiv_AufBahn <> eRolljobAufBahnPosiRuecklauf
		AND	strIO_GHdshk_Riem2.b_BahnZurueck )
	AND NOT strIO_GHdshk_Riem2.b_MTeilNichtFreigegeben
	AND NOT strIO_GLmHand.bI_QuittStoerung
	AND	bI_Automatik
	AND	bI_MitUeberwachungTeilNichtFreigegeben
THEN
	strIO_GHdshk_Riem2.b_MTeilNichtFreigegeben:= TRUE;

ELSIF	strIO_GLmHand.bI_QuittStoerung
THEN
	strIO_GHdshk_Riem2.b_MTeilNichtFreigegeben:= FALSE;
END_IF;
END_ACTION

ACTION Y_Struktur_Roll1:
(*----------------------------------------------------------------------------------------------------------------------------------*)
(*----------------------------------------------------------------------------------------------------------------------------------*)
(*                Struktur																		*)
(*----------------------------------------------------------------------------------------------------------------------------------*)
(*----------------------------------------------------------------------------------------------------------------------------------*)
strIO_GHdshk_Roll1.b_ExterneBahn						:= FALSE;
strIO_GHdshk_Roll1.b_LiAnfang							:= fbEntprellenAnfang_Roll1.OsSensor;
strIO_GHdshk_Roll1.b_SwAnfang							:= bSwAnfang_Roll1;
strIO_GHdshk_Roll1.b_LiVorAnfang						:= fbEntprellenVorAnfang_Roll1.OsSensor;
strIO_GHdshk_Roll1.b_SwVorAnfang						:= bSwVorAnfang_Roll1;
strIO_GHdshk_Roll1.b_LiEnde							:= fbEntprellenEnde_Roll1.OsSensor;
strIO_GHdshk_Roll1.b_SwEnde							:= bSwEnde_Roll1;
strIO_GHdshk_Roll1.b_LiVorEnde						:= fbEntprellenVorEnde_Roll1.OsSensor;
strIO_GHdshk_Roll1.b_SwVorEnde						:= bSwVorEnde_Roll1;
strIO_GHdshk_Roll1.b_LiBelegtkontrolle					:= fbEntprellenBelegtkontrolle_Roll1.OsSensor;
strIO_GHdshk_Roll1.b_BahnIstAufFoerderhoehe				:= fbBahn_Roll1.IsBahnIstAufFoerderhoehe;
strIO_GHdshk_Roll1.b_BahnVor							:= fbRampe_Roll1.bQ_MovePos;
strIO_GHdshk_Roll1.b_BahnZurueck						:= fbRampe_Roll1.bQ_MoveNeg;
strIO_GHdshk_Roll1.b_BahnSteht						:= fbRampe_Roll1.bQ_MoveNot;
strIO_GHdshk_Roll1.b_FreimeldungAnNachSektion				:= fbBahn_Roll1.OsFreimeldungAnNachSektion
												AND ( strIO_GHdshk_Roll1_Nachf.str_JobAktiv_VonBahn = eRollJobVonBahnRuecklauf
													OR	strIO_GHdshk_Roll1_Nachf.str_JobAktiv_VonBahn = eRollJobVonBahnPosiRuecklauf
													OR	strIO_GHdshk_Roll1_Nachf.b_SektionenKoppelnInX
													OR	strIO_GHdshk_Roll1_Nachf.b_SektionenKoppelnInY
													OR	strIO_GHdshk_Roll1_Nachf.b_ExterneBahn );
strIO_GHdshk_Roll1.b_FreimeldungAnVorSektion				:= fbBahn_Roll1.OsFreimeldungAnVorSektion
												AND ( strIO_GHdshk_Roll1_Vorg.str_JobAktiv_VonBahn = eRollJobVonBahnVorlauf
													OR	strIO_GHdshk_Roll1_Vorg.str_JobAktiv_VonBahn = eRollJobVonBahnPosiVorlauf
													OR	strIO_GHdshk_Roll1_Vorg.b_SektionenKoppelnInX
													OR	strIO_GHdshk_Roll1_Vorg.b_SektionenKoppelnInY
													OR	strIO_GHdshk_Roll1_Vorg.b_ExterneBahn );
strIO_GHdshk_Roll1.b_VerstandenPlatteAbgelegt				:= fbBahn_Roll1.OsVerstandenLaderPlatteAbgelegt;
strIO_GHdshk_Roll1.b_VerstandenPlatteGeholt				:= fbBahn_Roll1.OsVerstandenLaderPlatteGeholt;
strIO_GHdshk_Roll1.i_AblaufStatus_AufBahn					:= fbBahn_Roll1.OwAblaufStatus_AufBahn;
strIO_GHdshk_Roll1.i_AblaufStatus_VonBahn					:= fbBahn_Roll1.OwAblaufStatus_VonBahn;
strIO_GHdshk_Roll1.str_BahnStatus						:= fbBahn_Roll1.OwBahnStatus;
strIO_GHdshk_Roll1.str_JobAktiv_AufBahn					:= fbBahn_Roll1.OwJobAktiv_AufBahn;
strIO_GHdshk_Roll1.str_JobAktiv_VonBahn					:= fbBahn_Roll1.OwJobAktiv_VonBahn;
strIO_GHdshk_Roll1.b_MBahnBelegt_KeineDaten				:= fbBahn_Roll1.OsMBahnBelegt_KeineDaten;
strIO_GHdshk_Roll1.b_MBahnFrei_Daten					:= fbBahn_Roll1.OsMBahnFrei_Daten;
strIO_GHdshk_Roll1.b_MBahnNichtAufFoerderhoehe				:= fbBahn_Roll1.OsMBahnNichtAufFoerderhoehe;
strIO_GHdshk_Roll1.b_MMaxLaufzeit_AufBahn					:= fbBahn_Roll1.OsMMaxLaufzeit_AufBahn;
strIO_GHdshk_Roll1.b_MMaxLaufzeit_VonBahn					:= fbBahn_Roll1.OsMMaxLaufzeit_VonBahn;
strIO_GHdshk_Roll1.b_MStoerungAntrieb					:= fbBahn_Roll1.OsMStoerungAntrieb;
strIO_GHdshk_Roll1.b_MKeineFreigabe_FahrtInGrund			:= fbBahn_Roll1.OsMKeineFreigabe_FahrtInGrund;
strIO_GHdshk_Roll1.b_MFehlerRegisterimpuls				:= fbGeberKontrolle_Roll1.bQ_FehlerGeber;
strIO_GHdshk_Roll1.b_MFehlerSkalierung					:= fbGeberKontrolle_Roll1.bQ_FehlerSkalierung;

strIO_GHdshk_Roll1.b_GeberHandling_AufBahn_Aktiv			:= fbGeberHandling_AufBahn_Roll1.OsAktiv;
strIO_GHdshk_Roll1.b_GeberHandling_AufBahn_Fertig			:= fbGeberHandling_AufBahn_Roll1.OsFertig;
strIO_GHdshk_Roll1.r_PosiRestwert_AufBahn					:= fbGeberHandling_AufBahn_Roll1.OwPosiRestWert;

strIO_GHdshk_Roll1.b_GeberHandling_VonBahn_Aktiv			:= fbGeberHandling_VonBahn_Roll1.OsAktiv;
strIO_GHdshk_Roll1.b_GeberHandling_VonBahn_Fertig			:= fbGeberHandling_VonBahn_Roll1.OsFertig;
strIO_GHdshk_Roll1.r_PosiRestwert_VonBahn					:= fbGeberHandling_VonBahn_Roll1.OwPosiRestWert;

IF	fbRampe_Roll1.bI_Couple
THEN
	strIO_GHdshk_Roll1.lr_Bahnspeed_Soll				:= fbRampe_Roll1.lrI_CoupleVelocity;
ELSE
	strIO_GHdshk_Roll1.lr_Bahnspeed_Soll				:= fbRampe_Roll1.lrI_Velocity;
END_IF;

strIO_GHdshk_Roll1.lr_Bahnspeed_Vorgabe					:= fbRampe_Roll1.lrQ_ActVelocity;

IF	( strIO_GHdshk_Roll1.b_LiAnfang
	AND	strIO_GHdshk_Roll1.str_JobAktiv_AufBahn <> eRolljobAufBahnVorlauf
	AND	strIO_GHdshk_Roll1.str_JobAktiv_AufBahn <> eRolljobAufBahnPosiVorlauf
	AND	strIO_GHdshk_Roll1.b_BahnVor
	OR	strIO_GHdshk_Roll1.b_LiEnde
		AND	strIO_GHdshk_Roll1.str_JobAktiv_AufBahn <> eRolljobAufBahnRuecklauf
		AND	strIO_GHdshk_Roll1.str_JobAktiv_AufBahn <> eRolljobAufBahnPosiRuecklauf
		AND	strIO_GHdshk_Roll1.b_BahnZurueck )
	AND NOT strIO_GHdshk_Roll1.b_MTeilNichtFreigegeben
	AND NOT strIO_GLmHand.bI_QuittStoerung
	AND	bI_Automatik
	AND	bI_MitUeberwachungTeilNichtFreigegeben
THEN
	strIO_GHdshk_Roll1.b_MTeilNichtFreigegeben:= TRUE;

ELSIF	strIO_GLmHand.bI_QuittStoerung
THEN
	strIO_GHdshk_Roll1.b_MTeilNichtFreigegeben:= FALSE;
END_IF;
END_ACTION

ACTION Z_Meldungen_Riem1:
(*----------------------------------------------------------------------------------------------------------------------------------*)
(*----------------------------------------------------------------------------------------------------------------------------------*)
(*                Meldungen																		*)
(*----------------------------------------------------------------------------------------------------------------------------------*)
(*----------------------------------------------------------------------------------------------------------------------------------*)

(*0-4 Störung Antriebe*)
OfMeldung[uiI_FehlerId_Riem1+0]:= strIO_GHdshk_Riem1.b_MStoerungAntrieb;
OfMeldung[uiI_FehlerId_Riem1+1]:= FALSE;
OfMeldung[uiI_FehlerId_Riem1+2]:= FALSE;
OfMeldung[uiI_FehlerId_Riem1+3]:= FALSE;
OfMeldung[uiI_FehlerId_Riem1+4]:= FALSE;

(*5-9 Fehler Absoluter Stop*)
OfMeldung[uiI_FehlerId_Riem1+5]:= FALSE;
OfMeldung[uiI_FehlerId_Riem1+6]:= FALSE;
OfMeldung[uiI_FehlerId_Riem1+7]:= FALSE;
OfMeldung[uiI_FehlerId_Riem1+8]:= FALSE;
OfMeldung[uiI_FehlerId_Riem1+9]:= FALSE;

(*10-19 Fehler Bedingter Stop*)
OfMeldung[uiI_FehlerId_Riem1+10]:= fbRampe_Riem1.bQ_Error
						AND 	fbRampe_Riem1.uiQ_ErrorNumber = 100;
OfMeldung[uiI_FehlerId_Riem1+11]:= fbRampe_Riem1.bQ_Error
						AND 	fbRampe_Riem1.uiQ_ErrorNumber = 101;
OfMeldung[uiI_FehlerId_Riem1+12]:= fbRampe_Riem1.bQ_Error
						AND 	fbRampe_Riem1.uiQ_ErrorNumber = 102;
OfMeldung[uiI_FehlerId_Riem1+13]:= fbRampe_Riem1.bQ_Error
						AND 	fbRampe_Riem1.uiQ_ErrorNumber = 103;
OfMeldung[uiI_FehlerId_Riem1+14]:= fbRampe_Riem1.bQ_Error
						AND 	fbRampe_Riem1.uiQ_ErrorNumber = 104;
OfMeldung[uiI_FehlerId_Riem1+15]:= fbRampe_Riem1.bQ_Error
						AND 	fbRampe_Riem1.uiQ_ErrorNumber = 105;
OfMeldung[uiI_FehlerId_Riem1+16]:= FALSE;
OfMeldung[uiI_FehlerId_Riem1+17]:= FALSE;
OfMeldung[uiI_FehlerId_Riem1+18]:= FALSE;

IF	uiI_AxId_Riem1 > 0
THEN
	OfMeldung[uiI_FehlerId_Riem1+19]:= NOT AxFrNcGeeicht[uiI_AxId_Riem1];
ELSE
	OfMeldung[uiI_FehlerId_Riem1+19]:= FALSE;
END_IF;

